gfCNCPoint3[25201] = {X 315.6744, Y 14.7426, Z -4.6667, A 0.000, B 0.000, C 0.000 }
gfCNCPoint3[25202] = {X 315.1915, Y 15.5144, Z -4.6667, A 0.000, B 0.000, C 0.000 }
gfCNCPoint3[25203] = {X 314.5495, Y 16.1599, Z -4.6667, A 0.000, B 0.000, C 0.000 }
gfCNCPoint3[25204] = {X 314.5481, Y 41.0279, Z -4.6667, A 0.000, B 0.000, C 0.000 }
gfCNCPoint3[25205] = {X 314.6336, Y 41.0962, Z -4.6667, A 0.000, B 0.000, C 0.000 }
gfCNCPoint3[25206] = {X 315.2363, Y 41.7299, Z -4.6667, A 0.000, B 0.000, C 0.000 }
gfCNCPoint3[25207] = {X 315.6902, Y 42.4775, Z -4.6667, A 0.000, B 0.000, C 0.000 }
gfCNCPoint3[25208] = {X 315.9743, Y 43.3047, Z -4.6667, A 0.000, B 0.000, C 0.000 }
gfCNCPoint3[25209] = {X 316.0756, Y 44.1734, Z -4.6667, A 0.000, B 0.000, C 0.000 }
gfCNCPoint3[25210] = {X 316.0757, Y 45.0000, Z -4.6667, A 0.000, B 0.000, C 0.000 }
gfCNCPoint3[25211] = {X 315.9734, Y 45.9079, Z -4.6667, A 0.000, B 0.000, C 0.000 }
gfCNCPoint3[25212] = {X 315.6717, Y 46.7702, Z -4.6667, A 0.000, B 0.000, C 0.000 }
gfCNCPoint3[25213] = {X 315.1856, Y 47.5438, Z -4.6667, A 0.000, B 0.000, C 0.000 }
gfCNCPoint3[25214] = {X 314.5396, Y 48.1899, Z -4.6667, A 0.000, B 0.000, C 0.000 }
gfCNCPoint3[25215] = {X 313.7660, Y 48.6760, Z -4.6667, A 0.000, B 0.000, C 0.000 }
gfCNCPoint3[25216] = {X 312.9036, Y 48.9777, Z -4.6667, A 0.000, B 0.000, C 0.000 }
gfCNCPoint3[25217] = {X 311.9957, Y 49.0800, Z -4.6667, A 0.000, B 0.000, C 0.000 }
gfCNCPoint3[25218] = {X 305.5523, Y 49.0800, Z -4.6667, A 0.000, B 0.000, C 0.000 }
gfCNCPoint3[25219] = {X 304.6489, Y 48.9787, Z -4.6667, A 0.000, B 0.000, C 0.000 }
gfCNCPoint3[25220] = {X 303.7905, Y 48.6800, Z -4.6667, A 0.000, B 0.000, C 0.000 }
gfCNCPoint3[25221] = {X 303.0194, Y 48.1986, Z -4.6667, A 0.000, B 0.000, C 0.000 }
gfCNCPoint3[25222] = {X 302.3741, Y 47.5585, Z -4.6667, A 0.000, B 0.000, C 0.000 }
gfCNCPoint3[25223] = {X 301.8865, Y 46.7914, Z -4.6667, A 0.000, B 0.000, C 0.000 }
gfCNCPoint3[25224] = {X 301.5809, Y 45.9353, Z -4.6667, A 0.000, B 0.000, C 0.000 }
gfCNCPoint3[25225] = {X 301.4724, Y 45.0328, Z -4.6667, A 0.000, B 0.000, C 0.000 }
gfCNCPoint3[25226] = {X 301.4723, Y 44.2070, Z -4.6667, A 0.000, B 0.000, C 0.000 }
gfCNCPoint3[25227] = {X 301.5898, Y 43.2934, Z -4.6667, A 0.000, B 0.000, C 0.000 }
gfCNCPoint3[25228] = {X 301.8935, Y 42.4238, Z -4.6667, A 0.000, B 0.000, C 0.000 }
gfCNCPoint3[25229] = {X 302.3704, Y 41.6357, Z -4.6667, A 0.000, B 0.000, C 0.000 }
gfCNCPoint3[25230] = {X 302.9997, Y 40.9632, Z -4.6667, A 0.000, B 0.000, C 0.000 }
gfCNCPoint3[25231] = {X 302.9997, Y 33.7943, Z -4.6667, A 0.000, B 0.000, C 0.000 }
gfCNCPoint3[25232] = {X 293.6145, Y 33.7943, Z -4.6667, A 0.000, B 0.000, C 0.000 }
gfCNCPoint3[25233] = {X 293.6137, Y 41.0139, Z -4.6667, A 0.000, B 0.000, C 0.000 }
gfCNCPoint3[25234] = {X 294.2515, Y 41.6661, Z -4.6667, A 0.000, B 0.000, C 0.000 }
gfCNCPoint3[25235] = {X 294.7325, Y 42.4413, Z -4.6667, A 0.000, B 0.000, C 0.000 }
gfCNCPoint3[25236] = {X 295.0338, Y 43.3023, Z -4.6667, A 0.000, B 0.000, C 0.000 }
gfCNCPoint3[25237] = {X 295.1411, Y 44.2082, Z -4.6667, A 0.000, B 0.000, C 0.000 }
gfCNCPoint3[25238] = {X 295.1411, Y 45.0000, Z -4.6667, A 0.000, B 0.000, C 0.000 }
gfCNCPoint3[25239] = {X 295.0388, Y 45.9079, Z -4.6667, A 0.000, B 0.000, C 0.000 }
gfCNCPoint3[25240] = {X 294.7371, Y 46.7702, Z -4.6667, A 0.000, B 0.000, C 0.000 }
gfCNCPoint3[25241] = {X 294.2510, Y 47.5438, Z -4.6667, A 0.000, B 0.000, C 0.000 }
gfCNCPoint3[25242] = {X 293.6050, Y 48.1899, Z -4.6667, A 0.000, B 0.000, C 0.000 }
gfCNCPoint3[25243] = {X 292.8314, Y 48.6760, Z -4.6667, A 0.000, B 0.000, C 0.000 }
gfCNCPoint3[25244] = {X 291.9690, Y 48.9777, Z -4.6667, A 0.000, B 0.000, C 0.000 }
gfCNCPoint3[25245] = {X 291.0611, Y 49.0800, Z -4.6667, A 0.000, B 0.000, C 0.000 }
gfCNCPoint3[25246] = {X 284.6177, Y 49.0800, Z -4.6667, A 0.000, B 0.000, C 0.000 }
gfCNCPoint3[25247] = {X 283.7144, Y 48.9788, Z -4.6667, A 0.000, B 0.000, C 0.000 }
gfCNCPoint3[25248] = {X 282.8560, Y 48.6801, Z -4.6667, A 0.000, B 0.000, C 0.000 }
gfCNCPoint3[25249] = {X 282.0850, Y 48.1987, Z -4.6667, A 0.000, B 0.000, C 0.000 }
gfCNCPoint3[25250] = {X 281.4397, Y 47.5587, Z -4.6667, A 0.000, B 0.000, C 0.000 }
gfCNCPoint3[25251] = {X 280.9521, Y 46.7916, Z -4.6667, A 0.000, B 0.000, C 0.000 }
gfCNCPoint3[25252] = {X 280.6464, Y 45.9356, Z -4.6667, A 0.000, B 0.000, C 0.000 }
gfCNCPoint3[25253] = {X 280.5378, Y 45.0332, Z -4.6667, A 0.000, B 0.000, C 0.000 }
gfCNCPoint3[25254] = {X 280.5377, Y 44.2085, Z -4.6667, A 0.000, B 0.000, C 0.000 }
gfCNCPoint3[25255] = {X 280.6428, Y 43.3038, Z -4.6667, A 0.000, B 0.000, C 0.000 }
gfCNCPoint3[25256] = {X 280.9436, Y 42.4442, Z -4.6667, A 0.000, B 0.000, C 0.000 }
gfCNCPoint3[25257] = {X 281.4256, Y 41.6715, Z -4.6667, A 0.000, B 0.000, C 0.000 }
gfCNCPoint3[25258] = {X 282.0653, Y 41.0233, Z -4.6667, A 0.000, B 0.000, C 0.000 }
gfCNCPoint3[25259] = {X 282.0651, Y 28.5924, Z -4.6667, A 0.000, B 0.000, C 0.000 }
gfCNCPoint3[25260] = {X 278.0651, Y 28.5925, Z -4.6667, A 0.000, B 0.000, C 0.000 }
gfCNCPoint3[25261] = {X 282.1451, Y 28.5924, Z -4.6667, A 0.000, B 0.000, C 0.000 }
gfCNCPoint3[25262] = {X 282.1449, Y 16.1221, Z -4.6667, A 0.000, B 0.000, C 0.000 }
gfCNCPoint3[25263] = {X 281.5030, Y 15.4878, Z -4.6667, A 0.000, B 0.000, C 0.000 }
gfCNCPoint3[25264] = {X 281.0197, Y 14.7257, Z -4.6667, A 0.000, B 0.000, C 0.000 }
gfCNCPoint3[25265] = {X 280.7195, Y 13.8746, Z -4.6667, A 0.000, B 0.000, C 0.000 }
gfCNCPoint3[25266] = {X 280.6177, Y 12.9779, Z -4.6667, A 0.000, B 0.000, C 0.000 }
gfCNCPoint3[25267] = {X 280.6177, Y 12.1868, Z -4.6667, A 0.000, B 0.000, C 0.000 }
gfCNCPoint3[25268] = {X 280.7180, Y 11.2967, Z -4.6667, A 0.000, B 0.000, C 0.000 }
gfCNCPoint3[25269] = {X 281.0138, Y 10.4513, Z -4.6667, A 0.000, B 0.000, C 0.000 }
gfCNCPoint3[25270] = {X 281.4903, Y 9.6929, Z -4.6667, A 0.000, B 0.000, C 0.000 }
gfCNCPoint3[25271] = {X 282.1237, Y 9.0595, Z -4.6667, A 0.000, B 0.000, C 0.000 }
gfCNCPoint3[25272] = {X 282.8821, Y 8.5829, Z -4.6667, A 0.000, B 0.000, C 0.000 }
gfCNCPoint3[25273] = {X 283.7276, Y 8.2871, Z -4.6667, A 0.000, B 0.000, C 0.000 }
gfCNCPoint3[25274] = {X 284.6177, Y 8.1868, Z -4.6667, A 0.000, B 0.000, C 0.000 }
gfCNCPoint3[25275] = {X 291.0611, Y 8.1868, Z -4.6667, A 0.000, B 0.000, C 0.000 }
gfCNCPoint3[25276] = {X 291.9512, Y 8.2871, Z -4.6667, A 0.000, B 0.000, C 0.000 }
gfCNCPoint3[25277] = {X 292.7967, Y 8.5829, Z -4.6667, A 0.000, B 0.000, C 0.000 }
gfCNCPoint3[25278] = {X 293.5551, Y 9.0595, Z -4.6667, A 0.000, B 0.000, C 0.000 }
gfCNCPoint3[25279] = {X 294.1885, Y 9.6929, Z -4.6667, A 0.000, B 0.000, C 0.000 }
gfCNCPoint3[25280] = {X 294.6650, Y 10.4513, Z -4.6667, A 0.000, B 0.000, C 0.000 }
gfCNCPoint3[25281] = {X 294.9608, Y 11.2967, Z -4.6667, A 0.000, B 0.000, C 0.000 }
gfCNCPoint3[25282] = {X 295.0611, Y 12.1868, Z -4.6667, A 0.000, B 0.000, C 0.000 }
gfCNCPoint3[25283] = {X 295.0609, Y 13.0192, Z -4.6667, A 0.000, B 0.000, C 0.000 }
gfCNCPoint3[25284] = {X 294.9625, Y 13.8611, Z -4.6667, A 0.000, B 0.000, C 0.000 }
gfCNCPoint3[25285] = {X 294.6888, Y 14.6633, Z -4.6667, A 0.000, B 0.000, C 0.000 }
gfCNCPoint3[25286] = {X 294.2523, Y 15.3898, Z -4.6667, A 0.000, B 0.000, C 0.000 }
gfCNCPoint3[25287] = {X 293.6725, Y 16.0080, Z -4.6667, A 0.000, B 0.000, C 0.000 }
gfCNCPoint3[25288] = {X 293.5959, Y 16.0724, Z -4.6667, A 0.000, B 0.000, C 0.000 }
gfCNCPoint3[25289] = {X 293.5177, Y 16.1348, Z -4.6667, A 0.000, B 0.000, C 0.000 }
gfCNCPoint3[25290] = {X 293.5336, Y 16.1923, Z -4.6667, A 0.000, B 0.000, C 0.000 }
gfCNCPoint3[25291] = {X 293.5348, Y 22.5166, Z -4.6667, A 0.000, B 0.000, C 0.000 }
gfCNCPoint3[25292] = {X 293.7676, Y 22.5165, Z -4.6667, A 0.000, B 0.000, C 0.000 }
gfCNCPoint3[25293] = {X 303.0789, Y 22.5170, Z -4.6667, A 0.000, B 0.000, C 0.000 }
gfCNCPoint3[25294] = {X 303.0794, Y 16.1925, Z -4.6667, A 0.000, B 0.000, C 0.000 }
gfCNCPoint3[25295] = {X 303.0955, Y 16.1346, Z -4.6667, A 0.000, B 0.000, C 0.000 }
gfCNCPoint3[25296] = {X 303.0172, Y 16.0722, Z -4.6667, A 0.000, B 0.000, C 0.000 }
gfCNCPoint3[25297] = {X 302.9406, Y 16.0077, Z -4.6667, A 0.000, B 0.000, C 0.000 }
gfCNCPoint3[25298] = {X 302.3547, Y 15.3813, Z -4.6667, A 0.000, B 0.000, C 0.000 }
gfCNCPoint3[25299] = {X 301.9158, Y 14.6443, Z -4.6667, A 0.000, B 0.000, C 0.000 }
gfCNCPoint3[25300] = {X 301.6442, Y 13.8307, Z -4.6667, A 0.000, B 0.000, C 0.000 }
gfCNCPoint3[25301] = {X 301.5523, Y 12.9779, Z -4.6667, A 0.000, B 0.000, C 0.000 }
gfCNCPoint3[25302] = {X 301.5523, Y 12.1868, Z -4.6667, A 0.000, B 0.000, C 0.000 }
gfCNCPoint3[25303] = {X 301.6525, Y 11.2967, Z -4.6667, A 0.000, B 0.000, C 0.000 }
gfCNCPoint3[25304] = {X 301.9484, Y 10.4513, Z -4.6667, A 0.000, B 0.000, C 0.000 }
gfCNCPoint3[25305] = {X 302.4249, Y 9.6929, Z -4.6667, A 0.000, B 0.000, C 0.000 }
gfCNCPoint3[25306] = {X 303.0583, Y 9.0595, Z -4.6667, A 0.000, B 0.000, C 0.000 }
gfCNCPoint3[25307] = {X 303.8167, Y 8.5829, Z -4.6667, A 0.000, B 0.000, C 0.000 }
gfCNCPoint3[25308] = {X 304.6622, Y 8.2871, Z -4.6667, A 0.000, B 0.000, C 0.000 }
gfCNCPoint3[25309] = {X 305.5523, Y 8.1868, Z -4.6667, A 0.000, B 0.000, C 0.000 }
gfCNCPoint3[25310] = {X 311.9957, Y 8.1868, Z -4.6667, A 0.000, B 0.000, C 0.000 }
gfCNCPoint3[25311] = {X 312.8858, Y 8.2871, Z -4.6667, A 0.000, B 0.000, C 0.000 }
gfCNCPoint3[25312] = {X 313.7313, Y 8.5829, Z -4.6667, A 0.000, B 0.000, C 0.000 }
gfCNCPoint3[25313] = {X 314.4897, Y 9.0595, Z -4.6667, A 0.000, B 0.000, C 0.000 }
gfCNCPoint3[25314] = {X 315.1230, Y 9.6929, Z -4.6667, A 0.000, B 0.000, C 0.000 }
gfCNCPoint3[25315] = {X 315.5996, Y 10.4513, Z -4.6667, A 0.000, B 0.000, C 0.000 }
gfCNCPoint3[25316] = {X 315.8954, Y 11.2967, Z -4.6667, A 0.000, B 0.000, C 0.000 }
gfCNCPoint3[25317] = {X 315.9957, Y 12.1868, Z -4.6667, A 0.000, B 0.000, C 0.000 }
gfCNCPoint3[25318] = {X 315.9955, Y 13.0192, Z -4.6667, A 0.000, B 0.000, C 0.000 }
gfCNCPoint3[25319] = {X 315.8870, Y 13.9044, Z -4.6667, A 0.000, B 0.000, C 0.000 }
gfCNCPoint3[25320] = {X 315.5850, Y 14.7436, Z -4.6667, A 0.000, B 0.000, C 0.000 }
gfCNCPoint3[25321] = {X 315.1045, Y 15.4950, Z -4.6667, A 0.000, B 0.000, C 0.000 }
gfCNCPoint3[25322] = {X 314.4695, Y 16.1213, Z -4.6667, A 0.000, B 0.000, C 0.000 }
gfCNCPoint3[25323] = {X 314.4681, Y 41.0664, Z -4.6667, A 0.000, B 0.000, C 0.000 }
gfCNCPoint3[25324] = {X 314.6070, Y 41.1787, Z -4.6667, A 0.000, B 0.000, C 0.000 }
gfCNCPoint3[25325] = {X 315.1930, Y 41.8052, Z -4.6667, A 0.000, B 0.000, C 0.000 }
gfCNCPoint3[25326] = {X 315.6320, Y 42.5423, Z -4.6667, A 0.000, B 0.000, C 0.000 }
gfCNCPoint3[25327] = {X 315.9038, Y 43.3560, Z -4.6667, A 0.000, B 0.000, C 0.000 }
gfCNCPoint3[25328] = {X 315.9957, Y 44.2089, Z -4.6667, A 0.000, B 0.000, C 0.000 }
gfCNCPoint3[25329] = {X 315.9957, Y 45.0000, Z -4.6667, A 0.000, B 0.000, C 0.000 }
gfCNCPoint3[25330] = {X 315.8954, Y 45.8901, Z -4.6667, A 0.000, B 0.000, C 0.000 }
gfCNCPoint3[25331] = {X 315.5996, Y 46.7355, Z -4.6667, A 0.000, B 0.000, C 0.000 }
gfCNCPoint3[25332] = {X 315.1230, Y 47.4940, Z -4.6667, A 0.000, B 0.000, C 0.000 }
gfCNCPoint3[25333] = {X 314.4897, Y 48.1273, Z -4.6667, A 0.000, B 0.000, C 0.000 }
gfCNCPoint3[25334] = {X 313.7313, Y 48.6039, Z -4.6667, A 0.000, B 0.000, C 0.000 }
gfCNCPoint3[25335] = {X 312.8858, Y 48.8997, Z -4.6667, A 0.000, B 0.000, C 0.000 }
gfCNCPoint3[25336] = {X 311.9957, Y 49.0000, Z -4.6667, A 0.000, B 0.000, C 0.000 }
gfCNCPoint3[25337] = {X 305.5523, Y 49.0000, Z -4.6667, A 0.000, B 0.000, C 0.000 }
gfCNCPoint3[25338] = {X 304.6622, Y 48.8997, Z -4.6667, A 0.000, B 0.000, C 0.000 }
gfCNCPoint3[25339] = {X 303.8167, Y 48.6039, Z -4.6667, A 0.000, B 0.000, C 0.000 }
gfCNCPoint3[25340] = {X 303.0583, Y 48.1273, Z -4.6667, A 0.000, B 0.000, C 0.000 }
gfCNCPoint3[25341] = {X 302.4249, Y 47.4939, Z -4.6667, A 0.000, B 0.000, C 0.000 }
gfCNCPoint3[25342] = {X 301.9484, Y 46.7355, Z -4.6667, A 0.000, B 0.000, C 0.000 }
gfCNCPoint3[25343] = {X 301.6525, Y 45.8901, Z -4.6667, A 0.000, B 0.000, C 0.000 }
gfCNCPoint3[25344] = {X 301.5523, Y 45.0000, Z -4.6667, A 0.000, B 0.000, C 0.000 }
gfCNCPoint3[25345] = {X 301.5523, Y 44.2089, Z -4.6667, A 0.000, B 0.000, C 0.000 }
gfCNCPoint3[25346] = {X 301.6698, Y 43.3029, Z -4.6667, A 0.000, B 0.000, C 0.000 }
gfCNCPoint3[25347] = {X 301.9737, Y 42.4414, Z -4.6667, A 0.000, B 0.000, C 0.000 }
gfCNCPoint3[25348] = {X 302.4507, Y 41.6623, Z -4.6667, A 0.000, B 0.000, C 0.000 }
gfCNCPoint3[25349] = {X 303.0797, Y 40.9999, Z -4.6667, A 0.000, B 0.000, C 0.000 }
gfCNCPoint3[25350] = {X 303.0797, Y 33.7143, Z -4.6667, A 0.000, B 0.000, C 0.000 }
gfCNCPoint3[25351] = {X 293.9345, Y 33.7143, Z -4.6667, A 0.000, B 0.000, C 0.000 }
gfCNCPoint3[25352] = {X 293.5345, Y 33.7139, Z -4.6667, A 0.000, B 0.000, C 0.000 }
gfCNCPoint3[25353] = {X 293.5337, Y 41.0520, Z -4.6667, A 0.000, B 0.000, C 0.000 }
gfCNCPoint3[25354] = {X 294.1710, Y 41.6933, Z -4.6667, A 0.000, B 0.000, C 0.000 }
gfCNCPoint3[25355] = {X 294.6521, Y 42.4588, Z -4.6667, A 0.000, B 0.000, C 0.000 }
gfCNCPoint3[25356] = {X 294.9538, Y 43.3111, Z -4.6667, A 0.000, B 0.000, C 0.000 }
gfCNCPoint3[25357] = {X 295.0611, Y 44.2089, Z -4.6667, A 0.000, B 0.000, C 0.000 }
gfCNCPoint3[25358] = {X 295.0611, Y 45.0000, Z -4.6667, A 0.000, B 0.000, C 0.000 }
gfCNCPoint3[25359] = {X 294.9608, Y 45.8901, Z -4.6667, A 0.000, B 0.000, C 0.000 }
gfCNCPoint3[25360] = {X 294.6650, Y 46.7355, Z -4.6667, A 0.000, B 0.000, C 0.000 }
gfCNCPoint3[25361] = {X 294.1885, Y 47.4940, Z -4.6667, A 0.000, B 0.000, C 0.000 }
gfCNCPoint3[25362] = {X 293.5551, Y 48.1273, Z -4.6667, A 0.000, B 0.000, C 0.000 }
gfCNCPoint3[25363] = {X 292.7967, Y 48.6039, Z -4.6667, A 0.000, B 0.000, C 0.000 }
gfCNCPoint3[25364] = {X 291.9512, Y 48.8997, Z -4.6667, A 0.000, B 0.000, C 0.000 }
gfCNCPoint3[25365] = {X 291.0611, Y 49.0000, Z -4.6667, A 0.000, B 0.000, C 0.000 }
gfCNCPoint3[25366] = {X 284.6177, Y 49.0000, Z -4.6667, A 0.000, B 0.000, C 0.000 }
gfCNCPoint3[25367] = {X 283.7276, Y 48.8997, Z -4.6667, A 0.000, B 0.000, C 0.000 }
gfCNCPoint3[25368] = {X 282.8821, Y 48.6039, Z -4.6667, A 0.000, B 0.000, C 0.000 }
gfCNCPoint3[25369] = {X 282.1237, Y 48.1273, Z -4.6667, A 0.000, B 0.000, C 0.000 }
gfCNCPoint3[25370] = {X 281.4903, Y 47.4939, Z -4.6667, A 0.000, B 0.000, C 0.000 }
gfCNCPoint3[25371] = {X 281.0138, Y 46.7355, Z -4.6667, A 0.000, B 0.000, C 0.000 }
gfCNCPoint3[25372] = {X 280.7180, Y 45.8901, Z -4.6667, A 0.000, B 0.000, C 0.000 }
gfCNCPoint3[25373] = {X 280.6177, Y 45.0000, Z -4.6667, A 0.000, B 0.000, C 0.000 }
gfCNCPoint3[25374] = {X 280.6177, Y 44.2089, Z -4.6667, A 0.000, B 0.000, C 0.000 }
gfCNCPoint3[25375] = {X 280.7229, Y 43.3125, Z -4.6667, A 0.000, B 0.000, C 0.000 }
gfCNCPoint3[25376] = {X 281.0240, Y 42.4617, Z -4.6667, A 0.000, B 0.000, C 0.000 }
gfCNCPoint3[25377] = {X 281.5062, Y 41.6988, Z -4.6667, A 0.000, B 0.000, C 0.000 }
gfCNCPoint3[25378] = {X 282.1453, Y 41.0616, Z -4.6667, A 0.000, B 0.000, C 0.000 }
gfCNCPoint3[25379] = {X 282.1451, Y 28.5924, Z -4.6667, A 0.000, B 0.000, C 0.000 }
gfCNCPoint3[25380] = {X 278.0651, Y 28.5925, Z -4.6667, A 0.000, B 0.000, C 0.000 }
gfCNCPoint3[25381] = {X 278.0651, Y 28.5925, Z -1.6667, A 0.000, B 0.000, C 0.000 }
gfCNCPoint3[25382] = {X 278.0651, Y 28.5925, Z 11.0000, A 0.000, B 0.000, C 0.000 }
gfCNCPoint3[25383] = {X 353.3541, Y 107.0405, Z 11.0000, A 0.000, B 0.000, C 0.000 }
gfCNCPoint3[25384] = {X 353.3541, Y 107.0405, Z -1.6667, A 0.000, B 0.000, C 0.000 }
gfCNCPoint3[25385] = {X 353.3541, Y 107.0405, Z -4.6667, A 0.000, B 0.000, C 0.000 }
gfCNCPoint3[25386] = {X 353.2427, Y 102.9621, Z -4.6667, A 0.000, B 0.000, C 0.000 }
gfCNCPoint3[25387] = {X 348.1840, Y 103.0319, Z -4.6667, A 0.000, B 0.000, C 0.000 }
gfCNCPoint3[25388] = {X 343.1252, Y 102.9652, Z -4.6667, A 0.000, B 0.000, C 0.000 }
gfCNCPoint3[25389] = {X 338.0701, Y 102.7618, Z -4.6667, A 0.000, B 0.000, C 0.000 }
gfCNCPoint3[25390] = {X 334.1158, Y 102.4849, Z -4.6667, A 0.000, B 0.000, C 0.000 }
gfCNCPoint3[25391] = {X 330.1765, Y 102.0430, Z -4.6667, A 0.000, B 0.000, C 0.000 }
gfCNCPoint3[25392] = {X 326.2591, Y 101.4370, Z -4.6667, A 0.000, B 0.000, C 0.000 }
gfCNCPoint3[25393] = {X 323.4092, Y 100.8331, Z -4.6667, A 0.000, B 0.000, C 0.000 }
gfCNCPoint3[25394] = {X 320.6117, Y 100.0201, Z -4.6667, A 0.000, B 0.000, C 0.000 }
gfCNCPoint3[25395] = {X 317.8820, Y 99.0025, Z -4.6667, A 0.000, B 0.000, C 0.000 }
gfCNCPoint3[25396] = {X 316.3696, Y 98.3039, Z -4.6667, A 0.000, B 0.000, C 0.000 }
gfCNCPoint3[25397] = {X 314.9207, Y 97.4819, Z -4.6667, A 0.000, B 0.000, C 0.000 }
gfCNCPoint3[25398] = {X 313.5452, Y 96.5421, Z -4.6667, A 0.000, B 0.000, C 0.000 }
gfCNCPoint3[25399] = {X 312.2527, Y 95.4911, Z -4.6667, A 0.000, B 0.000, C 0.000 }
gfCNCPoint3[25400] = {X 311.2489, Y 94.4926, Z -4.6667, A 0.000, B 0.000, C 0.000 }
gfCNCPoint3[25401] = {X 310.3706, Y 93.3822, Z -4.6667, A 0.000, B 0.000, C 0.000 }
gfCNCPoint3[25402] = {X 309.6302, Y 92.1754, Z -4.6667, A 0.000, B 0.000, C 0.000 }
gfCNCPoint3[25403] = {X 309.0381, Y 90.8894, Z -4.6667, A 0.000, B 0.000, C 0.000 }
gfCNCPoint3[25404] = {X 308.6026, Y 89.5423, Z -4.6667, A 0.000, B 0.000, C 0.000 }
gfCNCPoint3[25405] = {X 308.2592, Y 87.9192, Z -4.6667, A 0.000, B 0.000, C 0.000 }
gfCNCPoint3[25406] = {X 308.0563, Y 86.2726, Z -4.6667, A 0.000, B 0.000, C 0.000 }
gfCNCPoint3[25407] = {X 307.9954, Y 84.6147, Z -4.6667, A 0.000, B 0.000, C 0.000 }
gfCNCPoint3[25408] = {X 307.9966, Y 63.2123, Z -4.6667, A 0.000, B 0.000, C 0.000 }
gfCNCPoint3[25409] = {X 307.1451, Y 63.0030, Z -4.6667, A 0.000, B 0.000, C 0.000 }
gfCNCPoint3[25410] = {X 306.3533, Y 62.6262, Z -4.6667, A 0.000, B 0.000, C 0.000 }
gfCNCPoint3[25411] = {X 305.6540, Y 62.0972, Z -4.6667, A 0.000, B 0.000, C 0.000 }
gfCNCPoint3[25412] = {X 305.0759, Y 61.4379, Z -4.6667, A 0.000, B 0.000, C 0.000 }
gfCNCPoint3[25413] = {X 304.6428, Y 60.6755, Z -4.6667, A 0.000, B 0.000, C 0.000 }
gfCNCPoint3[25414] = {X 304.3726, Y 59.8413, Z -4.6667, A 0.000, B 0.000, C 0.000 }
gfCNCPoint3[25415] = {X 304.2764, Y 58.9697, Z -4.6667, A 0.000, B 0.000, C 0.000 }
gfCNCPoint3[25416] = {X 304.2762, Y 58.0000, Z -4.6667, A 0.000, B 0.000, C 0.000 }
gfCNCPoint3[25417] = {X 304.3845, Y 57.0387, Z -4.6667, A 0.000, B 0.000, C 0.000 }
gfCNCPoint3[25418] = {X 304.7040, Y 56.1256, Z -4.6667, A 0.000, B 0.000, C 0.000 }
gfCNCPoint3[25419] = {X 305.2187, Y 55.3065, Z -4.6667, A 0.000, B 0.000, C 0.000 }
gfCNCPoint3[25420] = {X 305.9027, Y 54.6225, Z -4.6667, A 0.000, B 0.000, C 0.000 }
gfCNCPoint3[25421] = {X 306.7218, Y 54.1078, Z -4.6667, A 0.000, B 0.000, C 0.000 }
gfCNCPoint3[25422] = {X 307.6349, Y 53.7883, Z -4.6667, A 0.000, B 0.000, C 0.000 }
gfCNCPoint3[25423] = {X 308.5962, Y 53.6800, Z -4.6667, A 0.000, B 0.000, C 0.000 }
gfCNCPoint3[25424] = {X 324.3107, Y 53.6800, Z -4.6667, A 0.000, B 0.000, C 0.000 }
gfCNCPoint3[25425] = {X 325.2720, Y 53.7883, Z -4.6667, A 0.000, B 0.000, C 0.000 }
gfCNCPoint3[25426] = {X 326.1851, Y 54.1078, Z -4.6667, A 0.000, B 0.000, C 0.000 }
gfCNCPoint3[25427] = {X 327.0042, Y 54.6225, Z -4.6667, A 0.000, B 0.000, C 0.000 }
gfCNCPoint3[25428] = {X 327.6882, Y 55.3065, Z -4.6667, A 0.000, B 0.000, C 0.000 }
gfCNCPoint3[25429] = {X 328.2029, Y 56.1256, Z -4.6667, A 0.000, B 0.000, C 0.000 }
gfCNCPoint3[25430] = {X 328.5224, Y 57.0387, Z -4.6667, A 0.000, B 0.000, C 0.000 }
gfCNCPoint3[25431] = {X 328.6307, Y 58.0000, Z -4.6667, A 0.000, B 0.000, C 0.000 }
gfCNCPoint3[25432] = {X 328.6307, Y 58.9359, Z -4.6667, A 0.000, B 0.000, C 0.000 }
gfCNCPoint3[25433] = {X 328.5366, Y 59.8122, Z -4.6667, A 0.000, B 0.000, C 0.000 }
gfCNCPoint3[25434] = {X 328.2681, Y 60.6516, Z -4.6667, A 0.000, B 0.000, C 0.000 }
gfCNCPoint3[25435] = {X 327.8362, Y 61.4199, Z -4.6667, A 0.000, B 0.000, C 0.000 }
gfCNCPoint3[25436] = {X 327.2587, Y 62.0856, Z -4.6667, A 0.000, B 0.000, C 0.000 }
gfCNCPoint3[25437] = {X 326.5590, Y 62.6214, Z -4.6667, A 0.000, B 0.000, C 0.000 }
gfCNCPoint3[25438] = {X 325.7658, Y 63.0056, Z -4.6667, A 0.000, B 0.000, C 0.000 }
gfCNCPoint3[25439] = {X 324.9116, Y 63.2223, Z -4.6667, A 0.000, B 0.000, C 0.000 }
gfCNCPoint3[25440] = {X 324.9132, Y 83.2295, Z -4.6667, A 0.000, B 0.000, C 0.000 }
gfCNCPoint3[25441] = {X 324.9268, Y 84.6147, Z -4.6667, A 0.000, B 0.000, C 0.000 }
gfCNCPoint3[25442] = {X 325.0042, Y 85.8499, Z -4.6667, A 0.000, B 0.000, C 0.000 }
gfCNCPoint3[25443] = {X 325.2261, Y 87.0674, Z -4.6667, A 0.000, B 0.000, C 0.000 }
gfCNCPoint3[25444] = {X 325.4715, Y 87.3361, Z -4.6667, A 0.000, B 0.000, C 0.000 }
gfCNCPoint3[25445] = {X 325.7737, Y 87.5389, Z -4.6667, A 0.000, B 0.000, C 0.000 }
gfCNCPoint3[25446] = {X 326.2246, Y 87.7937, Z -4.6667, A 0.000, B 0.000, C 0.000 }
gfCNCPoint3[25447] = {X 327.6624, Y 88.3904, Z -4.6667, A 0.000, B 0.000, C 0.000 }
gfCNCPoint3[25448] = {X 329.1569, Y 88.8260, Z -4.6667, A 0.000, B 0.000, C 0.000 }
gfCNCPoint3[25449] = {X 332.2329, Y 89.4419, Z -4.6667, A 0.000, B 0.000, C 0.000 }
gfCNCPoint3[25450] = {X 335.3453, Y 89.8349, Z -4.6667, A 0.000, B 0.000, C 0.000 }
gfCNCPoint3[25451] = {X 339.4834, Y 90.1549, Z -4.6667, A 0.000, B 0.000, C 0.000 }
gfCNCPoint3[25452] = {X 343.6300, Y 90.3344, Z -4.6667, A 0.000, B 0.000, C 0.000 }
gfCNCPoint3[25453] = {X 347.7803, Y 90.3734, Z -4.6667, A 0.000, B 0.000, C 0.000 }
gfCNCPoint3[25454] = {X 352.1620, Y 90.3350, Z -4.6667, A 0.000, B 0.000, C 0.000 }
gfCNCPoint3[25455] = {X 356.5395, Y 90.1391, Z -4.6667, A 0.000, B 0.000, C 0.000 }
gfCNCPoint3[25456] = {X 360.9071, Y 89.7860, Z -4.6667, A 0.000, B 0.000, C 0.000 }
gfCNCPoint3[25457] = {X 363.2212, Y 89.4982, Z -4.6667, A 0.000, B 0.000, C 0.000 }
gfCNCPoint3[25458] = {X 365.5139, Y 89.0719, Z -4.6667, A 0.000, B 0.000, C 0.000 }
gfCNCPoint3[25459] = {X 367.7768, Y 88.5085, Z -4.6667, A 0.000, B 0.000, C 0.000 }
gfCNCPoint3[25460] = {X 368.7087, Y 88.1952, Z -4.6667, A 0.000, B 0.000, C 0.000 }
gfCNCPoint3[25461] = {X 369.5996, Y 87.7794, Z -4.6667, A 0.000, B 0.000, C 0.000 }
gfCNCPoint3[25462] = {X 370.4383, Y 87.2663, Z -4.6667, A 0.000, B 0.000, C 0.000 }
gfCNCPoint3[25463] = {X 370.5880, Y 87.1105, Z -4.6667, A 0.000, B 0.000, C 0.000 }
gfCNCPoint3[25464] = {X 370.6652, Y 86.9086, Z -4.6667, A 0.000, B 0.000, C 0.000 }
gfCNCPoint3[25465] = {X 370.8563, Y 85.3737, Z -4.6667, A 0.000, B 0.000, C 0.000 }
gfCNCPoint3[25466] = {X 370.9201, Y 83.8283, Z -4.6667, A 0.000, B 0.000, C 0.000 }
gfCNCPoint3[25467] = {X 370.9205, Y 63.2124, Z -4.6667, A 0.000, B 0.000, C 0.000 }
gfCNCPoint3[25468] = {X 370.0688, Y 63.0033, Z -4.6667, A 0.000, B 0.000, C 0.000 }
gfCNCPoint3[25469] = {X 369.2769, Y 62.6265, Z -4.6667, A 0.000, B 0.000, C 0.000 }
gfCNCPoint3[25470] = {X 368.5774, Y 62.0975, Z -4.6667, A 0.000, B 0.000, C 0.000 }
gfCNCPoint3[25471] = {X 367.9991, Y 61.4382, Z -4.6667, A 0.000, B 0.000, C 0.000 }
gfCNCPoint3[25472] = {X 367.5659, Y 60.6757, Z -4.6667, A 0.000, B 0.000, C 0.000 }
gfCNCPoint3[25473] = {X 367.2956, Y 59.8414, Z -4.6667, A 0.000, B 0.000, C 0.000 }
gfCNCPoint3[25474] = {X 367.1994, Y 58.9697, Z -4.6667, A 0.000, B 0.000, C 0.000 }
gfCNCPoint3[25475] = {X 367.1993, Y 58.0000, Z -4.6667, A 0.000, B 0.000, C 0.000 }
gfCNCPoint3[25476] = {X 367.3076, Y 57.0387, Z -4.6667, A 0.000, B 0.000, C 0.000 }
gfCNCPoint3[25477] = {X 367.6271, Y 56.1256, Z -4.6667, A 0.000, B 0.000, C 0.000 }
gfCNCPoint3[25478] = {X 368.1418, Y 55.3065, Z -4.6667, A 0.000, B 0.000, C 0.000 }
gfCNCPoint3[25479] = {X 368.8258, Y 54.6225, Z -4.6667, A 0.000, B 0.000, C 0.000 }
gfCNCPoint3[25480] = {X 369.6449, Y 54.1078, Z -4.6667, A 0.000, B 0.000, C 0.000 }
gfCNCPoint3[25481] = {X 370.5580, Y 53.7883, Z -4.6667, A 0.000, B 0.000, C 0.000 }
gfCNCPoint3[25482] = {X 371.5193, Y 53.6800, Z -4.6667, A 0.000, B 0.000, C 0.000 }
gfCNCPoint3[25483] = {X 388.0597, Y 53.6800, Z -4.6667, A 0.000, B 0.000, C 0.000 }
gfCNCPoint3[25484] = {X 389.0210, Y 53.7883, Z -4.6667, A 0.000, B 0.000, C 0.000 }
gfCNCPoint3[25485] = {X 389.9341, Y 54.1078, Z -4.6667, A 0.000, B 0.000, C 0.000 }
gfCNCPoint3[25486] = {X 390.7532, Y 54.6225, Z -4.6667, A 0.000, B 0.000, C 0.000 }
gfCNCPoint3[25487] = {X 391.4372, Y 55.3065, Z -4.6667, A 0.000, B 0.000, C 0.000 }
gfCNCPoint3[25488] = {X 391.9519, Y 56.1256, Z -4.6667, A 0.000, B 0.000, C 0.000 }
gfCNCPoint3[25489] = {X 392.2714, Y 57.0387, Z -4.6667, A 0.000, B 0.000, C 0.000 }
gfCNCPoint3[25490] = {X 392.3797, Y 58.0000, Z -4.6667, A 0.000, B 0.000, C 0.000 }
gfCNCPoint3[25491] = {X 392.3797, Y 58.9342, Z -4.6667, A 0.000, B 0.000, C 0.000 }
gfCNCPoint3[25492] = {X 392.2660, Y 59.9188, Z -4.6667, A 0.000, B 0.000, C 0.000 }
gfCNCPoint3[25493] = {X 391.9308, Y 60.8515, Z -4.6667, A 0.000, B 0.000, C 0.000 }
gfCNCPoint3[25494] = {X 391.4879, Y 61.5648, Z -4.6667, A 0.000, B 0.000, C 0.000 }
gfCNCPoint3[25495] = {X 390.9159, Y 62.1796, Z -4.6667, A 0.000, B 0.000, C 0.000 }
gfCNCPoint3[25496] = {X 390.2363, Y 62.6728, Z -4.6667, A 0.000, B 0.000, C 0.000 }
gfCNCPoint3[25497] = {X 389.4745, Y 63.0259, Z -4.6667, A 0.000, B 0.000, C 0.000 }
gfCNCPoint3[25498] = {X 388.6590, Y 63.2259, Z -4.6667, A 0.000, B 0.000, C 0.000 }
gfCNCPoint3[25499] = {X 388.6569, Y 84.6147, Z -4.6667, A 0.000, B 0.000, C 0.000 }
gfCNCPoint3[25500] = {X 388.5970, Y 86.2730, Z -4.6667, A 0.000, B 0.000, C 0.000 }
gfCNCPoint3[25501] = {X 388.3927, Y 87.9198, Z -4.6667, A 0.000, B 0.000, C 0.000 }
gfCNCPoint3[25502] = {X 388.0455, Y 89.5426, Z -4.6667, A 0.000, B 0.000, C 0.000 }
gfCNCPoint3[25503] = {X 387.5133, Y 91.1299, Z -4.6667, A 0.000, B 0.000, C 0.000 }
gfCNCPoint3[25504] = {X 386.7638, Y 92.6268, Z -4.6667, A 0.000, B 0.000, C 0.000 }
gfCNCPoint3[25505] = {X 385.8117, Y 94.0039, Z -4.6667, A 0.000, B 0.000, C 0.000 }
gfCNCPoint3[25506] = {X 384.6758, Y 95.2338, Z -4.6667, A 0.000, B 0.000, C 0.000 }
gfCNCPoint3[25507] = {X 383.1614, Y 96.5099, Z -4.6667, A 0.000, B 0.000, C 0.000 }
gfCNCPoint3[25508] = {X 381.5201, Y 97.6180, Z -4.6667, A 0.000, B 0.000, C 0.000 }
gfCNCPoint3[25509] = {X 379.7703, Y 98.5456, Z -4.6667, A 0.000, B 0.000, C 0.000 }
gfCNCPoint3[25510] = {X 377.4991, Y 99.5017, Z -4.6667, A 0.000, B 0.000, C 0.000 }
gfCNCPoint3[25511] = {X 375.1651, Y 100.2920, Z -4.6667, A 0.000, B 0.000, C 0.000 }
gfCNCPoint3[25512] = {X 372.7802, Y 100.9123, Z -4.6667, A 0.000, B 0.000, C 0.000 }
gfCNCPoint3[25513] = {X 368.8695, Y 101.6664, Z -4.6667, A 0.000, B 0.000, C 0.000 }
gfCNCPoint3[25514] = {X 364.9264, Y 102.2267, Z -4.6667, A 0.000, B 0.000, C 0.000 }
gfCNCPoint3[25515] = {X 360.9605, Y 102.5918, Z -4.6667, A 0.000, B 0.000, C 0.000 }
gfCNCPoint3[25516] = {X 357.1035, Y 102.8167, Z -4.6667, A 0.000, B 0.000, C 0.000 }
gfCNCPoint3[25517] = {X 353.2427, Y 102.9621, Z -4.6667, A 0.000, B 0.000, C 0.000 }
gfCNCPoint3[25518] = {X 353.3519, Y 106.9606, Z -4.6667, A 0.000, B 0.000, C 0.000 }
gfCNCPoint3[25519] = {X 353.2405, Y 102.8821, Z -4.6667, A 0.000, B 0.000, C 0.000 }
gfCNCPoint3[25520] = {X 348.1839, Y 102.9519, Z -4.6667, A 0.000, B 0.000, C 0.000 }
gfCNCPoint3[25521] = {X 343.1272, Y 102.8852, Z -4.6667, A 0.000, B 0.000, C 0.000 }
gfCNCPoint3[25522] = {X 338.0742, Y 102.6819, Z -4.6667, A 0.000, B 0.000, C 0.000 }
gfCNCPoint3[25523] = {X 334.1232, Y 102.4052, Z -4.6667, A 0.000, B 0.000, C 0.000 }
gfCNCPoint3[25524] = {X 330.1871, Y 101.9637, Z -4.6667, A 0.000, B 0.000, C 0.000 }
gfCNCPoint3[25525] = {X 326.2729, Y 101.3582, Z -4.6667, A 0.000, B 0.000, C 0.000 }
gfCNCPoint3[25526] = {X 323.4287, Y 100.7555, Z -4.6667, A 0.000, B 0.000, C 0.000 }
gfCNCPoint3[25527] = {X 320.6369, Y 99.9442, Z -4.6667, A 0.000, B 0.000, C 0.000 }
gfCNCPoint3[25528] = {X 317.9126, Y 98.9286, Z -4.6667, A 0.000, B 0.000, C 0.000 }
gfCNCPoint3[25529] = {X 316.4063, Y 98.2328, Z -4.6667, A 0.000, B 0.000, C 0.000 }
gfCNCPoint3[25530] = {X 314.9631, Y 97.4140, Z -4.6667, A 0.000, B 0.000, C 0.000 }
gfCNCPoint3[25531] = {X 313.5931, Y 96.4780, Z -4.6667, A 0.000, B 0.000, C 0.000 }
gfCNCPoint3[25532] = {X 312.3057, Y 95.4312, Z -4.6667, A 0.000, B 0.000, C 0.000 }
gfCNCPoint3[25533] = {X 311.3086, Y 94.4394, Z -4.6667, A 0.000, B 0.000, C 0.000 }
gfCNCPoint3[25534] = {X 310.4362, Y 93.3364, Z -4.6667, A 0.000, B 0.000, C 0.000 }
gfCNCPoint3[25535] = {X 309.7008, Y 92.1378, Z -4.6667, A 0.000, B 0.000, C 0.000 }
gfCNCPoint3[25536] = {X 309.1126, Y 90.8604, Z -4.6667, A 0.000, B 0.000, C 0.000 }
gfCNCPoint3[25537] = {X 308.6801, Y 89.5222, Z -4.6667, A 0.000, B 0.000, C 0.000 }
gfCNCPoint3[25538] = {X 308.3380, Y 87.9058, Z -4.6667, A 0.000, B 0.000, C 0.000 }
gfCNCPoint3[25539] = {X 308.1360, Y 86.2660, Z -4.6667, A 0.000, B 0.000, C 0.000 }
gfCNCPoint3[25540] = {X 308.0754, Y 84.6150, Z -4.6667, A 0.000, B 0.000, C 0.000 }
gfCNCPoint3[25541] = {X 308.0766, Y 63.1421, Z -4.6667, A 0.000, B 0.000, C 0.000 }
gfCNCPoint3[25542] = {X 307.2282, Y 62.9473, Z -4.6667, A 0.000, B 0.000, C 0.000 }
gfCNCPoint3[25543] = {X 306.4374, Y 62.5833, Z -4.6667, A 0.000, B 0.000, C 0.000 }
gfCNCPoint3[25544] = {X 305.7377, Y 62.0656, Z -4.6667, A 0.000, B 0.000, C 0.000 }
gfCNCPoint3[25545] = {X 305.1584, Y 61.4158, Z -4.6667, A 0.000, B 0.000, C 0.000 }
gfCNCPoint3[25546] = {X 304.7240, Y 60.6614, Z -4.6667, A 0.000, B 0.000, C 0.000 }
gfCNCPoint3[25547] = {X 304.4529, Y 59.8342, Z -4.6667, A 0.000, B 0.000, C 0.000 }
gfCNCPoint3[25548] = {X 304.3564, Y 58.9691, Z -4.6667, A 0.000, B 0.000, C 0.000 }
gfCNCPoint3[25549] = {X 304.3562, Y 58.0000, Z -4.6667, A 0.000, B 0.000, C 0.000 }
gfCNCPoint3[25550] = {X 304.4625, Y 57.0565, Z -4.6667, A 0.000, B 0.000, C 0.000 }
gfCNCPoint3[25551] = {X 304.7761, Y 56.1603, Z -4.6667, A 0.000, B 0.000, C 0.000 }
gfCNCPoint3[25552] = {X 305.2813, Y 55.3564, Z -4.6667, A 0.000, B 0.000, C 0.000 }
gfCNCPoint3[25553] = {X 305.9526, Y 54.6850, Z -4.6667, A 0.000, B 0.000, C 0.000 }
gfCNCPoint3[25554] = {X 306.7566, Y 54.1799, Z -4.6667, A 0.000, B 0.000, C 0.000 }
gfCNCPoint3[25555] = {X 307.6527, Y 53.8663, Z -4.6667, A 0.000, B 0.000, C 0.000 }
gfCNCPoint3[25556] = {X 308.5962, Y 53.7600, Z -4.6667, A 0.000, B 0.000, C 0.000 }
gfCNCPoint3[25557] = {X 324.3107, Y 53.7600, Z -4.6667, A 0.000, B 0.000, C 0.000 }
gfCNCPoint3[25558] = {X 325.2542, Y 53.8663, Z -4.6667, A 0.000, B 0.000, C 0.000 }
gfCNCPoint3[25559] = {X 326.1504, Y 54.1799, Z -4.6667, A 0.000, B 0.000, C 0.000 }
gfCNCPoint3[25560] = {X 326.9543, Y 54.6850, Z -4.6667, A 0.000, B 0.000, C 0.000 }
gfCNCPoint3[25561] = {X 327.6257, Y 55.3564, Z -4.6667, A 0.000, B 0.000, C 0.000 }
gfCNCPoint3[25562] = {X 328.1308, Y 56.1603, Z -4.6667, A 0.000, B 0.000, C 0.000 }
gfCNCPoint3[25563] = {X 328.4444, Y 57.0565, Z -4.6667, A 0.000, B 0.000, C 0.000 }
gfCNCPoint3[25564] = {X 328.5507, Y 58.0000, Z -4.6667, A 0.000, B 0.000, C 0.000 }
gfCNCPoint3[25565] = {X 328.5507, Y 58.9355, Z -4.6667, A 0.000, B 0.000, C 0.000 }
gfCNCPoint3[25566] = {X 328.4562, Y 59.8053, Z -4.6667, A 0.000, B 0.000, C 0.000 }
gfCNCPoint3[25567] = {X 328.1868, Y 60.6377, Z -4.6667, A 0.000, B 0.000, C 0.000 }
gfCNCPoint3[25568] = {X 327.7537, Y 61.3979, Z -4.6667, A 0.000, B 0.000, C 0.000 }
gfCNCPoint3[25569] = {X 327.1750, Y 62.0541, Z -4.6667, A 0.000, B 0.000, C 0.000 }
gfCNCPoint3[25570] = {X 326.4750, Y 62.5789, Z -4.6667, A 0.000, B 0.000, C 0.000 }
gfCNCPoint3[25571] = {X 325.6827, Y 62.9503, Z -4.6667, A 0.000, B 0.000, C 0.000 }
gfCNCPoint3[25572] = {X 324.8316, Y 63.1528, Z -4.6667, A 0.000, B 0.000, C 0.000 }
gfCNCPoint3[25573] = {X 324.8332, Y 83.2300, Z -4.6667, A 0.000, B 0.000, C 0.000 }
gfCNCPoint3[25574] = {X 324.8468, Y 84.6150, Z -4.6667, A 0.000, B 0.000, C 0.000 }
gfCNCPoint3[25575] = {X 324.9257, Y 85.8671, Z -4.6667, A 0.000, B 0.000, C 0.000 }
gfCNCPoint3[25576] = {X 325.1520, Y 87.1012, Z -4.6667, A 0.000, B 0.000, C 0.000 }
gfCNCPoint3[25577] = {X 325.4128, Y 87.3910, Z -4.6667, A 0.000, B 0.000, C 0.000 }
gfCNCPoint3[25578] = {X 325.7358, Y 87.6093, Z -4.6667, A 0.000, B 0.000, C 0.000 }
gfCNCPoint3[25579] = {X 326.1875, Y 87.8647, Z -4.6667, A 0.000, B 0.000, C 0.000 }
gfCNCPoint3[25580] = {X 327.6346, Y 88.4654, Z -4.6667, A 0.000, B 0.000, C 0.000 }
gfCNCPoint3[25581] = {X 329.1388, Y 88.9039, Z -4.6667, A 0.000, B 0.000, C 0.000 }
gfCNCPoint3[25582] = {X 332.2203, Y 89.5209, Z -4.6667, A 0.000, B 0.000, C 0.000 }
gfCNCPoint3[25583] = {X 335.3382, Y 89.9146, Z -4.6667, A 0.000, B 0.000, C 0.000 }
gfCNCPoint3[25584] = {X 339.4789, Y 90.2347, Z -4.6667, A 0.000, B 0.000, C 0.000 }
gfCNCPoint3[25585] = {X 343.6280, Y 90.4144, Z -4.6667, A 0.000, B 0.000, C 0.000 }
gfCNCPoint3[25586] = {X 347.7809, Y 90.4534, Z -4.6667, A 0.000, B 0.000, C 0.000 }
gfCNCPoint3[25587] = {X 352.1650, Y 90.4149, Z -4.6667, A 0.000, B 0.000, C 0.000 }
gfCNCPoint3[25588] = {X 356.5449, Y 90.2189, Z -4.6667, A 0.000, B 0.000, C 0.000 }
gfCNCPoint3[25589] = {X 360.9150, Y 89.8657, Z -4.6667, A 0.000, B 0.000, C 0.000 }
gfCNCPoint3[25590] = {X 363.2338, Y 89.5773, Z -4.6667, A 0.000, B 0.000, C 0.000 }
gfCNCPoint3[25591] = {X 365.5310, Y 89.1500, Z -4.6667, A 0.000, B 0.000, C 0.000 }
gfCNCPoint3[25592] = {X 367.7985, Y 88.5855, Z -4.6667, A 0.000, B 0.000, C 0.000 }
gfCNCPoint3[25593] = {X 368.7387, Y 88.2694, Z -4.6667, A 0.000, B 0.000, C 0.000 }
gfCNCPoint3[25594] = {X 369.6376, Y 87.8498, Z -4.6667, A 0.000, B 0.000, C 0.000 }
gfCNCPoint3[25595] = {X 370.4838, Y 87.3321, Z -4.6667, A 0.000, B 0.000, C 0.000 }
gfCNCPoint3[25596] = {X 370.6556, Y 87.1533, Z -4.6667, A 0.000, B 0.000, C 0.000 }
gfCNCPoint3[25597] = {X 370.7441, Y 86.9218, Z -4.6667, A 0.000, B 0.000, C 0.000 }
gfCNCPoint3[25598] = {X 370.9360, Y 85.3803, Z -4.6667, A 0.000, B 0.000, C 0.000 }
gfCNCPoint3[25599] = {X 371.0001, Y 83.8283, Z -4.6667, A 0.000, B 0.000, C 0.000 }
gfCNCPoint3[25600] = {X 371.0005, Y 63.1422, Z -4.6667, A 0.000, B 0.000, C 0.000 }
gfCNCPoint3[25601] = {X 370.1519, Y 62.9475, Z -4.6667, A 0.000, B 0.000, C 0.000 }
gfCNCPoint3[25602] = {X 369.3610, Y 62.5836, Z -4.6667, A 0.000, B 0.000, C 0.000 }
gfCNCPoint3[25603] = {X 368.6611, Y 62.0659, Z -4.6667, A 0.000, B 0.000, C 0.000 }
gfCNCPoint3[25604] = {X 368.0817, Y 61.4161, Z -4.6667, A 0.000, B 0.000, C 0.000 }
gfCNCPoint3[25605] = {X 367.6472, Y 60.6616, Z -4.6667, A 0.000, B 0.000, C 0.000 }
gfCNCPoint3[25606] = {X 367.3760, Y 59.8343, Z -4.6667, A 0.000, B 0.000, C 0.000 }
gfCNCPoint3[25607] = {X 367.2794, Y 58.9691, Z -4.6667, A 0.000, B 0.000, C 0.000 }
gfCNCPoint3[25608] = {X 367.2793, Y 58.0000, Z -4.6667, A 0.000, B 0.000, C 0.000 }
gfCNCPoint3[25609] = {X 367.3856, Y 57.0565, Z -4.6667, A 0.000, B 0.000, C 0.000 }
gfCNCPoint3[25610] = {X 367.6992, Y 56.1603, Z -4.6667, A 0.000, B 0.000, C 0.000 }
gfCNCPoint3[25611] = {X 368.2043, Y 55.3564, Z -4.6667, A 0.000, B 0.000, C 0.000 }
gfCNCPoint3[25612] = {X 368.8757, Y 54.6850, Z -4.6667, A 0.000, B 0.000, C 0.000 }
gfCNCPoint3[25613] = {X 369.6796, Y 54.1799, Z -4.6667, A 0.000, B 0.000, C 0.000 }
gfCNCPoint3[25614] = {X 370.5758, Y 53.8663, Z -4.6667, A 0.000, B 0.000, C 0.000 }
gfCNCPoint3[25615] = {X 371.5193, Y 53.7600, Z -4.6667, A 0.000, B 0.000, C 0.000 }
gfCNCPoint3[25616] = {X 388.0597, Y 53.7600, Z -4.6667, A 0.000, B 0.000, C 0.000 }
gfCNCPoint3[25617] = {X 389.0032, Y 53.8663, Z -4.6667, A 0.000, B 0.000, C 0.000 }
gfCNCPoint3[25618] = {X 389.8993, Y 54.1799, Z -4.6667, A 0.000, B 0.000, C 0.000 }
gfCNCPoint3[25619] = {X 390.7033, Y 54.6850, Z -4.6667, A 0.000, B 0.000, C 0.000 }
gfCNCPoint3[25620] = {X 391.3746, Y 55.3564, Z -4.6667, A 0.000, B 0.000, C 0.000 }
gfCNCPoint3[25621] = {X 391.8798, Y 56.1603, Z -4.6667, A 0.000, B 0.000, C 0.000 }
gfCNCPoint3[25622] = {X 392.1934, Y 57.0565, Z -4.6667, A 0.000, B 0.000, C 0.000 }
gfCNCPoint3[25623] = {X 392.2997, Y 58.0000, Z -4.6667, A 0.000, B 0.000, C 0.000 }
gfCNCPoint3[25624] = {X 392.2997, Y 58.9342, Z -4.6667, A 0.000, B 0.000, C 0.000 }
gfCNCPoint3[25625] = {X 392.1881, Y 59.9005, Z -4.6667, A 0.000, B 0.000, C 0.000 }
gfCNCPoint3[25626] = {X 391.8592, Y 60.8160, Z -4.6667, A 0.000, B 0.000, C 0.000 }
gfCNCPoint3[25627] = {X 391.4159, Y 61.5272, Z -4.6667, A 0.000, B 0.000, C 0.000 }
gfCNCPoint3[25628] = {X 390.8422, Y 62.1379, Z -4.6667, A 0.000, B 0.000, C 0.000 }
gfCNCPoint3[25629] = {X 390.1599, Y 62.6246, Z -4.6667, A 0.000, B 0.000, C 0.000 }
gfCNCPoint3[25630] = {X 389.3957, Y 62.9684, Z -4.6667, A 0.000, B 0.000, C 0.000 }
gfCNCPoint3[25631] = {X 388.5790, Y 63.1560, Z -4.6667, A 0.000, B 0.000, C 0.000 }
gfCNCPoint3[25632] = {X 388.5769, Y 84.6150, Z -4.6667, A 0.000, B 0.000, C 0.000 }
gfCNCPoint3[25633] = {X 388.5173, Y 86.2665, Z -4.6667, A 0.000, B 0.000, C 0.000 }
gfCNCPoint3[25634] = {X 388.3138, Y 87.9065, Z -4.6667, A 0.000, B 0.000, C 0.000 }
gfCNCPoint3[25635] = {X 387.9681, Y 89.5224, Z -4.6667, A 0.000, B 0.000, C 0.000 }
gfCNCPoint3[25636] = {X 387.4395, Y 91.0991, Z -4.6667, A 0.000, B 0.000, C 0.000 }
gfCNCPoint3[25637] = {X 386.6949, Y 92.5860, Z -4.6667, A 0.000, B 0.000, C 0.000 }
gfCNCPoint3[25638] = {X 385.7492, Y 93.9538, Z -4.6667, A 0.000, B 0.000, C 0.000 }
gfCNCPoint3[25639] = {X 384.6210, Y 95.1755, Z -4.6667, A 0.000, B 0.000, C 0.000 }
gfCNCPoint3[25640] = {X 383.1131, Y 96.4461, Z -4.6667, A 0.000, B 0.000, C 0.000 }
gfCNCPoint3[25641] = {X 381.4788, Y 97.5494, Z -4.6667, A 0.000, B 0.000, C 0.000 }
gfCNCPoint3[25642] = {X 379.7367, Y 98.4730, Z -4.6667, A 0.000, B 0.000, C 0.000 }
gfCNCPoint3[25643] = {X 377.4708, Y 99.4269, Z -4.6667, A 0.000, B 0.000, C 0.000 }
gfCNCPoint3[25644] = {X 375.1421, Y 100.2153, Z -4.6667, A 0.000, B 0.000, C 0.000 }
gfCNCPoint3[25645] = {X 372.7628, Y 100.8342, Z -4.6667, A 0.000, B 0.000, C 0.000 }
gfCNCPoint3[25646] = {X 368.8561, Y 101.5875, Z -4.6667, A 0.000, B 0.000, C 0.000 }
gfCNCPoint3[25647] = {X 364.9169, Y 102.1472, Z -4.6667, A 0.000, B 0.000, C 0.000 }
gfCNCPoint3[25648] = {X 360.9550, Y 102.5120, Z -4.6667, A 0.000, B 0.000, C 0.000 }
gfCNCPoint3[25649] = {X 357.0996, Y 102.7368, Z -4.6667, A 0.000, B 0.000, C 0.000 }
gfCNCPoint3[25650] = {X 353.2405, Y 102.8821, Z -4.6667, A 0.000, B 0.000, C 0.000 }
gfCNCPoint3[25651] = {X 353.3497, Y 106.8806, Z -4.6667, A 0.000, B 0.000, C 0.000 }
gfCNCPoint3[25652] = {X 353.2383, Y 102.8021, Z -4.6667, A 0.000, B 0.000, C 0.000 }
gfCNCPoint3[25653] = {X 348.1838, Y 102.8719, Z -4.6667, A 0.000, B 0.000, C 0.000 }
gfCNCPoint3[25654] = {X 343.1292, Y 102.8052, Z -4.6667, A 0.000, B 0.000, C 0.000 }
gfCNCPoint3[25655] = {X 338.0783, Y 102.6020, Z -4.6667, A 0.000, B 0.000, C 0.000 }
gfCNCPoint3[25656] = {X 334.1305, Y 102.3256, Z -4.6667, A 0.000, B 0.000, C 0.000 }
gfCNCPoint3[25657] = {X 330.1977, Y 101.8844, Z -4.6667, A 0.000, B 0.000, C 0.000 }
gfCNCPoint3[25658] = {X 326.2868, Y 101.2794, Z -4.6667, A 0.000, B 0.000, C 0.000 }
gfCNCPoint3[25659] = {X 323.4483, Y 100.6780, Z -4.6667, A 0.000, B 0.000, C 0.000 }
gfCNCPoint3[25660] = {X 320.6620, Y 99.8682, Z -4.6667, A 0.000, B 0.000, C 0.000 }
gfCNCPoint3[25661] = {X 317.9433, Y 98.8547, Z -4.6667, A 0.000, B 0.000, C 0.000 }
gfCNCPoint3[25662] = {X 316.4429, Y 98.1617, Z -4.6667, A 0.000, B 0.000, C 0.000 }
gfCNCPoint3[25663] = {X 315.0055, Y 97.3462, Z -4.6667, A 0.000, B 0.000, C 0.000 }
gfCNCPoint3[25664] = {X 313.6409, Y 96.4139, Z -4.6667, A 0.000, B 0.000, C 0.000 }
gfCNCPoint3[25665] = {X 312.3587, Y 95.3712, Z -4.6667, A 0.000, B 0.000, C 0.000 }
gfCNCPoint3[25666] = {X 311.3684, Y 94.3862, Z -4.6667, A 0.000, B 0.000, C 0.000 }
gfCNCPoint3[25667] = {X 310.5019, Y 93.2906, Z -4.6667, A 0.000, B 0.000, C 0.000 }
gfCNCPoint3[25668] = {X 309.7713, Y 92.1001, Z -4.6667, A 0.000, B 0.000, C 0.000 }
gfCNCPoint3[25669] = {X 309.1872, Y 90.8313, Z -4.6667, A 0.000, B 0.000, C 0.000 }
gfCNCPoint3[25670] = {X 308.7575, Y 89.5022, Z -4.6667, A 0.000, B 0.000, C 0.000 }
gfCNCPoint3[25671] = {X 308.4169, Y 87.8925, Z -4.6667, A 0.000, B 0.000, C 0.000 }
gfCNCPoint3[25672] = {X 308.2157, Y 86.2595, Z -4.6667, A 0.000, B 0.000, C 0.000 }
gfCNCPoint3[25673] = {X 308.1554, Y 84.6152, Z -4.6667, A 0.000, B 0.000, C 0.000 }
gfCNCPoint3[25674] = {X 308.1566, Y 63.0708, Z -4.6667, A 0.000, B 0.000, C 0.000 }
gfCNCPoint3[25675] = {X 307.3115, Y 62.8907, Z -4.6667, A 0.000, B 0.000, C 0.000 }
gfCNCPoint3[25676] = {X 306.5218, Y 62.5399, Z -4.6667, A 0.000, B 0.000, C 0.000 }
gfCNCPoint3[25677] = {X 305.8216, Y 62.0336, Z -4.6667, A 0.000, B 0.000, C 0.000 }
gfCNCPoint3[25678] = {X 305.2411, Y 61.3935, Z -4.6667, A 0.000, B 0.000, C 0.000 }
gfCNCPoint3[25679] = {X 304.8054, Y 60.6472, Z -4.6667, A 0.000, B 0.000, C 0.000 }
gfCNCPoint3[25680] = {X 304.5332, Y 59.8271, Z -4.6667, A 0.000, B 0.000, C 0.000 }
gfCNCPoint3[25681] = {X 304.4364, Y 58.9684, Z -4.6667, A 0.000, B 0.000, C 0.000 }
gfCNCPoint3[25682] = {X 304.4362, Y 58.0000, Z -4.6667, A 0.000, B 0.000, C 0.000 }
gfCNCPoint3[25683] = {X 304.5405, Y 57.0743, Z -4.6667, A 0.000, B 0.000, C 0.000 }
gfCNCPoint3[25684] = {X 304.8482, Y 56.1950, Z -4.6667, A 0.000, B 0.000, C 0.000 }
gfCNCPoint3[25685] = {X 305.3438, Y 55.4063, Z -4.6667, A 0.000, B 0.000, C 0.000 }
gfCNCPoint3[25686] = {X 306.0025, Y 54.7476, Z -4.6667, A 0.000, B 0.000, C 0.000 }
gfCNCPoint3[25687] = {X 306.7913, Y 54.2520, Z -4.6667, A 0.000, B 0.000, C 0.000 }
gfCNCPoint3[25688] = {X 307.6705, Y 53.9443, Z -4.6667, A 0.000, B 0.000, C 0.000 }
gfCNCPoint3[25689] = {X 308.5962, Y 53.8400, Z -4.6667, A 0.000, B 0.000, C 0.000 }
gfCNCPoint3[25690] = {X 324.3107, Y 53.8400, Z -4.6667, A 0.000, B 0.000, C 0.000 }
gfCNCPoint3[25691] = {X 325.2364, Y 53.9443, Z -4.6667, A 0.000, B 0.000, C 0.000 }
gfCNCPoint3[25692] = {X 326.1156, Y 54.2520, Z -4.6667, A 0.000, B 0.000, C 0.000 }
gfCNCPoint3[25693] = {X 326.9044, Y 54.7476, Z -4.6667, A 0.000, B 0.000, C 0.000 }
gfCNCPoint3[25694] = {X 327.5631, Y 55.4063, Z -4.6667, A 0.000, B 0.000, C 0.000 }
gfCNCPoint3[25695] = {X 328.0587, Y 56.1950, Z -4.6667, A 0.000, B 0.000, C 0.000 }
gfCNCPoint3[25696] = {X 328.3664, Y 57.0743, Z -4.6667, A 0.000, B 0.000, C 0.000 }
gfCNCPoint3[25697] = {X 328.4707, Y 58.0000, Z -4.6667, A 0.000, B 0.000, C 0.000 }
gfCNCPoint3[25698] = {X 328.4707, Y 58.9350, Z -4.6667, A 0.000, B 0.000, C 0.000 }
gfCNCPoint3[25699] = {X 328.3759, Y 59.7984, Z -4.6667, A 0.000, B 0.000, C 0.000 }
gfCNCPoint3[25700] = {X 328.1055, Y 60.6237, Z -4.6667, A 0.000, B 0.000, C 0.000 }
gfCNCPoint3[25701] = {X 327.6711, Y 61.3758, Z -4.6667, A 0.000, B 0.000, C 0.000 }
gfCNCPoint3[25702] = {X 327.0912, Y 62.0224, Z -4.6667, A 0.000, B 0.000, C 0.000 }
gfCNCPoint3[25703] = {X 326.3907, Y 62.5358, Z -4.6667, A 0.000, B 0.000, C 0.000 }
gfCNCPoint3[25704] = {X 325.5995, Y 62.8942, Z -4.6667, A 0.000, B 0.000, C 0.000 }
gfCNCPoint3[25705] = {X 324.7516, Y 63.0820, Z -4.6667, A 0.000, B 0.000, C 0.000 }
gfCNCPoint3[25706] = {X 324.7532, Y 83.2304, Z -4.6667, A 0.000, B 0.000, C 0.000 }
gfCNCPoint3[25707] = {X 324.7668, Y 84.6153, Z -4.6667, A 0.000, B 0.000, C 0.000 }
gfCNCPoint3[25708] = {X 324.8472, Y 85.8842, Z -4.6667, A 0.000, B 0.000, C 0.000 }
gfCNCPoint3[25709] = {X 325.0779, Y 87.1346, Z -4.6667, A 0.000, B 0.000, C 0.000 }
gfCNCPoint3[25710] = {X 325.3539, Y 87.4458, Z -4.6667, A 0.000, B 0.000, C 0.000 }
gfCNCPoint3[25711] = {X 325.6979, Y 87.6798, Z -4.6667, A 0.000, B 0.000, C 0.000 }
gfCNCPoint3[25712] = {X 326.1504, Y 87.9356, Z -4.6667, A 0.000, B 0.000, C 0.000 }
gfCNCPoint3[25713] = {X 327.6068, Y 88.5404, Z -4.6667, A 0.000, B 0.000, C 0.000 }
gfCNCPoint3[25714] = {X 329.1206, Y 88.9818, Z -4.6667, A 0.000, B 0.000, C 0.000 }
gfCNCPoint3[25715] = {X 332.2076, Y 89.5999, Z -4.6667, A 0.000, B 0.000, C 0.000 }
gfCNCPoint3[25716] = {X 335.3310, Y 89.9942, Z -4.6667, A 0.000, B 0.000, C 0.000 }
gfCNCPoint3[25717] = {X 339.4743, Y 90.3146, Z -4.6667, A 0.000, B 0.000, C 0.000 }
gfCNCPoint3[25718] = {X 343.6261, Y 90.4944, Z -4.6667, A 0.000, B 0.000, C 0.000 }
gfCNCPoint3[25719] = {X 347.7815, Y 90.5334, Z -4.6667, A 0.000, B 0.000, C 0.000 }
gfCNCPoint3[25720] = {X 352.1681, Y 90.4949, Z -4.6667, A 0.000, B 0.000, C 0.000 }
gfCNCPoint3[25721] = {X 356.5504, Y 90.2987, Z -4.6667, A 0.000, B 0.000, C 0.000 }
gfCNCPoint3[25722] = {X 360.9228, Y 89.9453, Z -4.6667, A 0.000, B 0.000, C 0.000 }
gfCNCPoint3[25723] = {X 363.2463, Y 89.6563, Z -4.6667, A 0.000, B 0.000, C 0.000 }
gfCNCPoint3[25724] = {X 365.5481, Y 89.2282, Z -4.6667, A 0.000, B 0.000, C 0.000 }
gfCNCPoint3[25725] = {X 367.8201, Y 88.6625, Z -4.6667, A 0.000, B 0.000, C 0.000 }
gfCNCPoint3[25726] = {X 368.7687, Y 88.3435, Z -4.6667, A 0.000, B 0.000, C 0.000 }
gfCNCPoint3[25727] = {X 369.6756, Y 87.9202, Z -4.6667, A 0.000, B 0.000, C 0.000 }
gfCNCPoint3[25728] = {X 370.5293, Y 87.3979, Z -4.6667, A 0.000, B 0.000, C 0.000 }
gfCNCPoint3[25729] = {X 370.7231, Y 87.1962, Z -4.6667, A 0.000, B 0.000, C 0.000 }
gfCNCPoint3[25730] = {X 370.8230, Y 86.9349, Z -4.6667, A 0.000, B 0.000, C 0.000 }
gfCNCPoint3[25731] = {X 371.0158, Y 85.3869, Z -4.6667, A 0.000, B 0.000, C 0.000 }
gfCNCPoint3[25732] = {X 371.0801, Y 83.8283, Z -4.6667, A 0.000, B 0.000, C 0.000 }
gfCNCPoint3[25733] = {X 371.0805, Y 63.0709, Z -4.6667, A 0.000, B 0.000, C 0.000 }
gfCNCPoint3[25734] = {X 370.9780, Y 63.0587, Z -4.6667, A 0.000, B 0.000, C 0.000 }
gfCNCPoint3[25735] = {X 370.8758, Y 63.0440, Z -4.6667, A 0.000, B 0.000, C 0.000 }
gfCNCPoint3[25736] = {X 369.9383, Y 62.7819, Z -4.6667, A 0.000, B 0.000, C 0.000 }
gfCNCPoint3[25737] = {X 369.0873, Y 62.3092, Z -4.6667, A 0.000, B 0.000, C 0.000 }
gfCNCPoint3[25738] = {X 368.3696, Y 61.6516, Z -4.6667, A 0.000, B 0.000, C 0.000 }
gfCNCPoint3[25739] = {X 367.8243, Y 60.8452, Z -4.6667, A 0.000, B 0.000, C 0.000 }
gfCNCPoint3[25740] = {X 367.4813, Y 59.9342, Z -4.6667, A 0.000, B 0.000, C 0.000 }
gfCNCPoint3[25741] = {X 367.3594, Y 58.9684, Z -4.6667, A 0.000, B 0.000, C 0.000 }
gfCNCPoint3[25742] = {X 367.3593, Y 58.0000, Z -4.6667, A 0.000, B 0.000, C 0.000 }
gfCNCPoint3[25743] = {X 367.4636, Y 57.0743, Z -4.6667, A 0.000, B 0.000, C 0.000 }
gfCNCPoint3[25744] = {X 367.7713, Y 56.1950, Z -4.6667, A 0.000, B 0.000, C 0.000 }
gfCNCPoint3[25745] = {X 368.2669, Y 55.4063, Z -4.6667, A 0.000, B 0.000, C 0.000 }
gfCNCPoint3[25746] = {X 368.9256, Y 54.7476, Z -4.6667, A 0.000, B 0.000, C 0.000 }
gfCNCPoint3[25747] = {X 369.7143, Y 54.2520, Z -4.6667, A 0.000, B 0.000, C 0.000 }
gfCNCPoint3[25748] = {X 370.5936, Y 53.9443, Z -4.6667, A 0.000, B 0.000, C 0.000 }
gfCNCPoint3[25749] = {X 371.5193, Y 53.8400, Z -4.6667, A 0.000, B 0.000, C 0.000 }
gfCNCPoint3[25750] = {X 388.0597, Y 53.8400, Z -4.6667, A 0.000, B 0.000, C 0.000 }
gfCNCPoint3[25751] = {X 388.9854, Y 53.9443, Z -4.6667, A 0.000, B 0.000, C 0.000 }
gfCNCPoint3[25752] = {X 389.8646, Y 54.2520, Z -4.6667, A 0.000, B 0.000, C 0.000 }
gfCNCPoint3[25753] = {X 390.6534, Y 54.7476, Z -4.6667, A 0.000, B 0.000, C 0.000 }
gfCNCPoint3[25754] = {X 391.3121, Y 55.4063, Z -4.6667, A 0.000, B 0.000, C 0.000 }
gfCNCPoint3[25755] = {X 391.8077, Y 56.1950, Z -4.6667, A 0.000, B 0.000, C 0.000 }
gfCNCPoint3[25756] = {X 392.1154, Y 57.0743, Z -4.6667, A 0.000, B 0.000, C 0.000 }
gfCNCPoint3[25757] = {X 392.2197, Y 58.0000, Z -4.6667, A 0.000, B 0.000, C 0.000 }
gfCNCPoint3[25758] = {X 392.2197, Y 58.9342, Z -4.6667, A 0.000, B 0.000, C 0.000 }
gfCNCPoint3[25759] = {X 392.1102, Y 59.8823, Z -4.6667, A 0.000, B 0.000, C 0.000 }
gfCNCPoint3[25760] = {X 391.7875, Y 60.7805, Z -4.6667, A 0.000, B 0.000, C 0.000 }
gfCNCPoint3[25761] = {X 391.2441, Y 61.6118, Z -4.6667, A 0.000, B 0.000, C 0.000 }
gfCNCPoint3[25762] = {X 390.5200, Y 62.2916, Z -4.6667, A 0.000, B 0.000, C 0.000 }
gfCNCPoint3[25763] = {X 389.6561, Y 62.7815, Z -4.6667, A 0.000, B 0.000, C 0.000 }
gfCNCPoint3[25764] = {X 388.7010, Y 63.0538, Z -4.6667, A 0.000, B 0.000, C 0.000 }
gfCNCPoint3[25765] = {X 388.6008, Y 63.0686, Z -4.6667, A 0.000, B 0.000, C 0.000 }
gfCNCPoint3[25766] = {X 388.5002, Y 63.0810, Z -4.6667, A 0.000, B 0.000, C 0.000 }
gfCNCPoint3[25767] = {X 388.4969, Y 84.6154, Z -4.6667, A 0.000, B 0.000, C 0.000 }
gfCNCPoint3[25768] = {X 388.4376, Y 86.2599, Z -4.6667, A 0.000, B 0.000, C 0.000 }
gfCNCPoint3[25769] = {X 388.2349, Y 87.8931, Z -4.6667, A 0.000, B 0.000, C 0.000 }
gfCNCPoint3[25770] = {X 387.8906, Y 89.5023, Z -4.6667, A 0.000, B 0.000, C 0.000 }
gfCNCPoint3[25771] = {X 387.3656, Y 91.0683, Z -4.6667, A 0.000, B 0.000, C 0.000 }
gfCNCPoint3[25772] = {X 386.6261, Y 92.5452, Z -4.6667, A 0.000, B 0.000, C 0.000 }
gfCNCPoint3[25773] = {X 385.6868, Y 93.9038, Z -4.6667, A 0.000, B 0.000, C 0.000 }
gfCNCPoint3[25774] = {X 384.5662, Y 95.1172, Z -4.6667, A 0.000, B 0.000, C 0.000 }
gfCNCPoint3[25775] = {X 383.0648, Y 96.3823, Z -4.6667, A 0.000, B 0.000, C 0.000 }
gfCNCPoint3[25776] = {X 381.4376, Y 97.4808, Z -4.6667, A 0.000, B 0.000, C 0.000 }
gfCNCPoint3[25777] = {X 379.7030, Y 98.4004, Z -4.6667, A 0.000, B 0.000, C 0.000 }
gfCNCPoint3[25778] = {X 377.4424, Y 99.3521, Z -4.6667, A 0.000, B 0.000, C 0.000 }
gfCNCPoint3[25779] = {X 375.1192, Y 100.1387, Z -4.6667, A 0.000, B 0.000, C 0.000 }
gfCNCPoint3[25780] = {X 372.7455, Y 100.7561, Z -4.6667, A 0.000, B 0.000, C 0.000 }
gfCNCPoint3[25781] = {X 368.8427, Y 101.5086, Z -4.6667, A 0.000, B 0.000, C 0.000 }
gfCNCPoint3[25782] = {X 364.9075, Y 102.0678, Z -4.6667, A 0.000, B 0.000, C 0.000 }
gfCNCPoint3[25783] = {X 360.9496, Y 102.4322, Z -4.6667, A 0.000, B 0.000, C 0.000 }
gfCNCPoint3[25784] = {X 357.0958, Y 102.6569, Z -4.6667, A 0.000, B 0.000, C 0.000 }
gfCNCPoint3[25785] = {X 353.2383, Y 102.8021, Z -4.6667, A 0.000, B 0.000, C 0.000 }
gfCNCPoint3[25786] = {X 353.3476, Y 106.8006, Z -4.6667, A 0.000, B 0.000, C 0.000 }
gfCNCPoint3[25787] = {X 353.2361, Y 102.7222, Z -4.6667, A 0.000, B 0.000, C 0.000 }
gfCNCPoint3[25788] = {X 348.1837, Y 102.7919, Z -4.6667, A 0.000, B 0.000, C 0.000 }
gfCNCPoint3[25789] = {X 343.1313, Y 102.7252, Z -4.6667, A 0.000, B 0.000, C 0.000 }
gfCNCPoint3[25790] = {X 338.0825, Y 102.5221, Z -4.6667, A 0.000, B 0.000, C 0.000 }
gfCNCPoint3[25791] = {X 334.1379, Y 102.2459, Z -4.6667, A 0.000, B 0.000, C 0.000 }
gfCNCPoint3[25792] = {X 330.2084, Y 101.8051, Z -4.6667, A 0.000, B 0.000, C 0.000 }
gfCNCPoint3[25793] = {X 326.3006, Y 101.2006, Z -4.6667, A 0.000, B 0.000, C 0.000 }
gfCNCPoint3[25794] = {X 323.4678, Y 100.6004, Z -4.6667, A 0.000, B 0.000, C 0.000 }
gfCNCPoint3[25795] = {X 320.6872, Y 99.7923, Z -4.6667, A 0.000, B 0.000, C 0.000 }
gfCNCPoint3[25796] = {X 317.9739, Y 98.7808, Z -4.6667, A 0.000, B 0.000, C 0.000 }
gfCNCPoint3[25797] = {X 316.4796, Y 98.0906, Z -4.6667, A 0.000, B 0.000, C 0.000 }
gfCNCPoint3[25798] = {X 315.0479, Y 97.2784, Z -4.6667, A 0.000, B 0.000, C 0.000 }
gfCNCPoint3[25799] = {X 313.6888, Y 96.3498, Z -4.6667, A 0.000, B 0.000, C 0.000 }
gfCNCPoint3[25800] = {X 312.4117, Y 95.3113, Z -4.6667, A 0.000, B 0.000, C 0.000 }
gfCNCPoint3[25801] = {X 311.4281, Y 94.3330, Z -4.6667, A 0.000, B 0.000, C 0.000 }
gfCNCPoint3[25802] = {X 310.5675, Y 93.2449, Z -4.6667, A 0.000, B 0.000, C 0.000 }
gfCNCPoint3[25803] = {X 309.8419, Y 92.0624, Z -4.6667, A 0.000, B 0.000, C 0.000 }
gfCNCPoint3[25804] = {X 309.2617, Y 90.8022, Z -4.6667, A 0.000, B 0.000, C 0.000 }
gfCNCPoint3[25805] = {X 308.8350, Y 89.4822, Z -4.6667, A 0.000, B 0.000, C 0.000 }
gfCNCPoint3[25806] = {X 308.4958, Y 87.8792, Z -4.6667, A 0.000, B 0.000, C 0.000 }
gfCNCPoint3[25807] = {X 308.2955, Y 86.2530, Z -4.6667, A 0.000, B 0.000, C 0.000 }
gfCNCPoint3[25808] = {X 308.2354, Y 84.6156, Z -4.6667, A 0.000, B 0.000, C 0.000 }
gfCNCPoint3[25809] = {X 308.2366, Y 62.9982, Z -4.6667, A 0.000, B 0.000, C 0.000 }
gfCNCPoint3[25810] = {X 307.3949, Y 62.8332, Z -4.6667, A 0.000, B 0.000, C 0.000 }
gfCNCPoint3[25811] = {X 306.6063, Y 62.4959, Z -4.6667, A 0.000, B 0.000, C 0.000 }
gfCNCPoint3[25812] = {X 305.9057, Y 62.0012, Z -4.6667, A 0.000, B 0.000, C 0.000 }
gfCNCPoint3[25813] = {X 305.3239, Y 61.3709, Z -4.6667, A 0.000, B 0.000, C 0.000 }
gfCNCPoint3[25814] = {X 304.8868, Y 60.6330, Z -4.6667, A 0.000, B 0.000, C 0.000 }
gfCNCPoint3[25815] = {X 304.6136, Y 59.8199, Z -4.6667, A 0.000, B 0.000, C 0.000 }
gfCNCPoint3[25816] = {X 304.5164, Y 58.9678, Z -4.6667, A 0.000, B 0.000, C 0.000 }
gfCNCPoint3[25817] = {X 304.5162, Y 58.0000, Z -4.6667, A 0.000, B 0.000, C 0.000 }
gfCNCPoint3[25818] = {X 304.6185, Y 57.0921, Z -4.6667, A 0.000, B 0.000, C 0.000 }
gfCNCPoint3[25819] = {X 304.9203, Y 56.2298, Z -4.6667, A 0.000, B 0.000, C 0.000 }
gfCNCPoint3[25820] = {X 305.4064, Y 55.4562, Z -4.6667, A 0.000, B 0.000, C 0.000 }
gfCNCPoint3[25821] = {X 306.0524, Y 54.8101, Z -4.6667, A 0.000, B 0.000, C 0.000 }
gfCNCPoint3[25822] = {X 306.8260, Y 54.3240, Z -4.6667, A 0.000, B 0.000, C 0.000 }
gfCNCPoint3[25823] = {X 307.6883, Y 54.0223, Z -4.6667, A 0.000, B 0.000, C 0.000 }
gfCNCPoint3[25824] = {X 308.5962, Y 53.9200, Z -4.6667, A 0.000, B 0.000, C 0.000 }
gfCNCPoint3[25825] = {X 324.3107, Y 53.9200, Z -4.6667, A 0.000, B 0.000, C 0.000 }
gfCNCPoint3[25826] = {X 325.2186, Y 54.0223, Z -4.6667, A 0.000, B 0.000, C 0.000 }
gfCNCPoint3[25827] = {X 326.0809, Y 54.3240, Z -4.6667, A 0.000, B 0.000, C 0.000 }
gfCNCPoint3[25828] = {X 326.8545, Y 54.8101, Z -4.6667, A 0.000, B 0.000, C 0.000 }
gfCNCPoint3[25829] = {X 327.5006, Y 55.4562, Z -4.6667, A 0.000, B 0.000, C 0.000 }
gfCNCPoint3[25830] = {X 327.9866, Y 56.2298, Z -4.6667, A 0.000, B 0.000, C 0.000 }
gfCNCPoint3[25831] = {X 328.2884, Y 57.0921, Z -4.6667, A 0.000, B 0.000, C 0.000 }
gfCNCPoint3[25832] = {X 328.3907, Y 58.0000, Z -4.6667, A 0.000, B 0.000, C 0.000 }
gfCNCPoint3[25833] = {X 328.3907, Y 58.9346, Z -4.6667, A 0.000, B 0.000, C 0.000 }
gfCNCPoint3[25834] = {X 328.2956, Y 59.7914, Z -4.6667, A 0.000, B 0.000, C 0.000 }
gfCNCPoint3[25835] = {X 328.0241, Y 60.6097, Z -4.6667, A 0.000, B 0.000, C 0.000 }
gfCNCPoint3[25836] = {X 327.5883, Y 61.3535, Z -4.6667, A 0.000, B 0.000, C 0.000 }
gfCNCPoint3[25837] = {X 327.0072, Y 61.9903, Z -4.6667, A 0.000, B 0.000, C 0.000 }
gfCNCPoint3[25838] = {X 326.3062, Y 62.4922, Z -4.6667, A 0.000, B 0.000, C 0.000 }
gfCNCPoint3[25839] = {X 325.5161, Y 62.8371, Z -4.6667, A 0.000, B 0.000, C 0.000 }
gfCNCPoint3[25840] = {X 324.6715, Y 63.0101, Z -4.6667, A 0.000, B 0.000, C 0.000 }
gfCNCPoint3[25841] = {X 324.6732, Y 83.2309, Z -4.6667, A 0.000, B 0.000, C 0.000 }
gfCNCPoint3[25842] = {X 324.6868, Y 84.6156, Z -4.6667, A 0.000, B 0.000, C 0.000 }
gfCNCPoint3[25843] = {X 324.7687, Y 85.9012, Z -4.6667, A 0.000, B 0.000, C 0.000 }
gfCNCPoint3[25844] = {X 325.0037, Y 87.1678, Z -4.6667, A 0.000, B 0.000, C 0.000 }
gfCNCPoint3[25845] = {X 325.2950, Y 87.5005, Z -4.6667, A 0.000, B 0.000, C 0.000 }
gfCNCPoint3[25846] = {X 325.6599, Y 87.7502, Z -4.6667, A 0.000, B 0.000, C 0.000 }
gfCNCPoint3[25847] = {X 326.1134, Y 88.0066, Z -4.6667, A 0.000, B 0.000, C 0.000 }
gfCNCPoint3[25848] = {X 327.5789, Y 88.6154, Z -4.6667, A 0.000, B 0.000, C 0.000 }
gfCNCPoint3[25849] = {X 329.1025, Y 89.0598, Z -4.6667, A 0.000, B 0.000, C 0.000 }
gfCNCPoint3[25850] = {X 332.1949, Y 89.6788, Z -4.6667, A 0.000, B 0.000, C 0.000 }
gfCNCPoint3[25851] = {X 335.3238, Y 90.0739, Z -4.6667, A 0.000, B 0.000, C 0.000 }
gfCNCPoint3[25852] = {X 339.4695, Y 90.3945, Z -4.6667, A 0.000, B 0.000, C 0.000 }
gfCNCPoint3[25853] = {X 343.6236, Y 90.5744, Z -4.6667, A 0.000, B 0.000, C 0.000 }
gfCNCPoint3[25854] = {X 347.7815, Y 90.6134, Z -4.6667, A 0.000, B 0.000, C 0.000 }
gfCNCPoint3[25855] = {X 352.1707, Y 90.5748, Z -4.6667, A 0.000, B 0.000, C 0.000 }
gfCNCPoint3[25856] = {X 356.5556, Y 90.3786, Z -4.6667, A 0.000, B 0.000, C 0.000 }
gfCNCPoint3[25857] = {X 360.9307, Y 90.0249, Z -4.6667, A 0.000, B 0.000, C 0.000 }
gfCNCPoint3[25858] = {X 363.2588, Y 89.7353, Z -4.6667, A 0.000, B 0.000, C 0.000 }
gfCNCPoint3[25859] = {X 365.5653, Y 89.3063, Z -4.6667, A 0.000, B 0.000, C 0.000 }
gfCNCPoint3[25860] = {X 367.8418, Y 88.7395, Z -4.6667, A 0.000, B 0.000, C 0.000 }
gfCNCPoint3[25861] = {X 368.7987, Y 88.4177, Z -4.6667, A 0.000, B 0.000, C 0.000 }
gfCNCPoint3[25862] = {X 369.7136, Y 87.9906, Z -4.6667, A 0.000, B 0.000, C 0.000 }
gfCNCPoint3[25863] = {X 370.5748, Y 87.4637, Z -4.6667, A 0.000, B 0.000, C 0.000 }
gfCNCPoint3[25864] = {X 370.7907, Y 87.2391, Z -4.6667, A 0.000, B 0.000, C 0.000 }
gfCNCPoint3[25865] = {X 370.9020, Y 86.9481, Z -4.6667, A 0.000, B 0.000, C 0.000 }
gfCNCPoint3[25866] = {X 371.0955, Y 85.3935, Z -4.6667, A 0.000, B 0.000, C 0.000 }
gfCNCPoint3[25867] = {X 371.1601, Y 83.8283, Z -4.6667, A 0.000, B 0.000, C 0.000 }
gfCNCPoint3[25868] = {X 371.1605, Y 62.9983, Z -4.6667, A 0.000, B 0.000, C 0.000 }
gfCNCPoint3[25869] = {X 371.0240, Y 62.9839, Z -4.6667, A 0.000, B 0.000, C 0.000 }
gfCNCPoint3[25870] = {X 370.8881, Y 62.9650, Z -4.6667, A 0.000, B 0.000, C 0.000 }
gfCNCPoint3[25871] = {X 369.9687, Y 62.7079, Z -4.6667, A 0.000, B 0.000, C 0.000 }
gfCNCPoint3[25872] = {X 369.1341, Y 62.2443, Z -4.6667, A 0.000, B 0.000, C 0.000 }
gfCNCPoint3[25873] = {X 368.4301, Y 61.5993, Z -4.6667, A 0.000, B 0.000, C 0.000 }
gfCNCPoint3[25874] = {X 367.8953, Y 60.8085, Z -4.6667, A 0.000, B 0.000, C 0.000 }
gfCNCPoint3[25875] = {X 367.5590, Y 59.9150, Z -4.6667, A 0.000, B 0.000, C 0.000 }
gfCNCPoint3[25876] = {X 367.4394, Y 58.9678, Z -4.6667, A 0.000, B 0.000, C 0.000 }
gfCNCPoint3[25877] = {X 367.4393, Y 58.0000, Z -4.6667, A 0.000, B 0.000, C 0.000 }
gfCNCPoint3[25878] = {X 367.5416, Y 57.0921, Z -4.6667, A 0.000, B 0.000, C 0.000 }
gfCNCPoint3[25879] = {X 367.8433, Y 56.2298, Z -4.6667, A 0.000, B 0.000, C 0.000 }
gfCNCPoint3[25880] = {X 368.3294, Y 55.4562, Z -4.6667, A 0.000, B 0.000, C 0.000 }
gfCNCPoint3[25881] = {X 368.9754, Y 54.8101, Z -4.6667, A 0.000, B 0.000, C 0.000 }
gfCNCPoint3[25882] = {X 369.7490, Y 54.3240, Z -4.6667, A 0.000, B 0.000, C 0.000 }
gfCNCPoint3[25883] = {X 370.6114, Y 54.0223, Z -4.6667, A 0.000, B 0.000, C 0.000 }
gfCNCPoint3[25884] = {X 371.5193, Y 53.9200, Z -4.6667, A 0.000, B 0.000, C 0.000 }
gfCNCPoint3[25885] = {X 388.0597, Y 53.9200, Z -4.6667, A 0.000, B 0.000, C 0.000 }
gfCNCPoint3[25886] = {X 388.9676, Y 54.0223, Z -4.6667, A 0.000, B 0.000, C 0.000 }
gfCNCPoint3[25887] = {X 389.8299, Y 54.3240, Z -4.6667, A 0.000, B 0.000, C 0.000 }
gfCNCPoint3[25888] = {X 390.6035, Y 54.8101, Z -4.6667, A 0.000, B 0.000, C 0.000 }
gfCNCPoint3[25889] = {X 391.2496, Y 55.4562, Z -4.6667, A 0.000, B 0.000, C 0.000 }
gfCNCPoint3[25890] = {X 391.7356, Y 56.2298, Z -4.6667, A 0.000, B 0.000, C 0.000 }
gfCNCPoint3[25891] = {X 392.0374, Y 57.0921, Z -4.6667, A 0.000, B 0.000, C 0.000 }
gfCNCPoint3[25892] = {X 392.1397, Y 58.0000, Z -4.6667, A 0.000, B 0.000, C 0.000 }
gfCNCPoint3[25893] = {X 392.1397, Y 58.9342, Z -4.6667, A 0.000, B 0.000, C 0.000 }
gfCNCPoint3[25894] = {X 392.0323, Y 59.8641, Z -4.6667, A 0.000, B 0.000, C 0.000 }
gfCNCPoint3[25895] = {X 391.7158, Y 60.7450, Z -4.6667, A 0.000, B 0.000, C 0.000 }
gfCNCPoint3[25896] = {X 391.1828, Y 61.5604, Z -4.6667, A 0.000, B 0.000, C 0.000 }
gfCNCPoint3[25897] = {X 390.4726, Y 62.2272, Z -4.6667, A 0.000, B 0.000, C 0.000 }
gfCNCPoint3[25898] = {X 389.6252, Y 62.7077, Z -4.6667, A 0.000, B 0.000, C 0.000 }
gfCNCPoint3[25899] = {X 388.6884, Y 62.9748, Z -4.6667, A 0.000, B 0.000, C 0.000 }
gfCNCPoint3[25900] = {X 388.5551, Y 62.9939, Z -4.6667, A 0.000, B 0.000, C 0.000 }
gfCNCPoint3[25901] = {X 388.4213, Y 63.0087, Z -4.6667, A 0.000, B 0.000, C 0.000 }
gfCNCPoint3[25902] = {X 388.4190, Y 63.1547, Z -4.6667, A 0.000, B 0.000, C 0.000 }
gfCNCPoint3[25903] = {X 388.4169, Y 84.6157, Z -4.6667, A 0.000, B 0.000, C 0.000 }
gfCNCPoint3[25904] = {X 388.3578, Y 86.2534, Z -4.6667, A 0.000, B 0.000, C 0.000 }
gfCNCPoint3[25905] = {X 388.1561, Y 87.8797, Z -4.6667, A 0.000, B 0.000, C 0.000 }
gfCNCPoint3[25906] = {X 387.8132, Y 89.4822, Z -4.6667, A 0.000, B 0.000, C 0.000 }
gfCNCPoint3[25907] = {X 387.2918, Y 91.0375, Z -4.6667, A 0.000, B 0.000, C 0.000 }
gfCNCPoint3[25908] = {X 386.5573, Y 92.5044, Z -4.6667, A 0.000, B 0.000, C 0.000 }
gfCNCPoint3[25909] = {X 385.6244, Y 93.8538, Z -4.6667, A 0.000, B 0.000, C 0.000 }
gfCNCPoint3[25910] = {X 384.5114, Y 95.0589, Z -4.6667, A 0.000, B 0.000, C 0.000 }
gfCNCPoint3[25911] = {X 383.0165, Y 96.3185, Z -4.6667, A 0.000, B 0.000, C 0.000 }
gfCNCPoint3[25912] = {X 381.3964, Y 97.4123, Z -4.6667, A 0.000, B 0.000, C 0.000 }
gfCNCPoint3[25913] = {X 379.6693, Y 98.3279, Z -4.6667, A 0.000, B 0.000, C 0.000 }
gfCNCPoint3[25914] = {X 377.4141, Y 99.2773, Z -4.6667, A 0.000, B 0.000, C 0.000 }
gfCNCPoint3[25915] = {X 375.0963, Y 100.0620, Z -4.6667, A 0.000, B 0.000, C 0.000 }
gfCNCPoint3[25916] = {X 372.7282, Y 100.6780, Z -4.6667, A 0.000, B 0.000, C 0.000 }
gfCNCPoint3[25917] = {X 368.8293, Y 101.4298, Z -4.6667, A 0.000, B 0.000, C 0.000 }
gfCNCPoint3[25918] = {X 364.8981, Y 101.9883, Z -4.6667, A 0.000, B 0.000, C 0.000 }
gfCNCPoint3[25919] = {X 360.9441, Y 102.3524, Z -4.6667, A 0.000, B 0.000, C 0.000 }
gfCNCPoint3[25920] = {X 357.0920, Y 102.5770, Z -4.6667, A 0.000, B 0.000, C 0.000 }
gfCNCPoint3[25921] = {X 353.2361, Y 102.7222, Z -4.6667, A 0.000, B 0.000, C 0.000 }
gfCNCPoint3[25922] = {X 353.3454, Y 106.7207, Z -4.6667, A 0.000, B 0.000, C 0.000 }
gfCNCPoint3[25923] = {X 353.2339, Y 102.6422, Z -4.6667, A 0.000, B 0.000, C 0.000 }
gfCNCPoint3[25924] = {X 348.1836, Y 102.7119, Z -4.6667, A 0.000, B 0.000, C 0.000 }
gfCNCPoint3[25925] = {X 343.1333, Y 102.6453, Z -4.6667, A 0.000, B 0.000, C 0.000 }
gfCNCPoint3[25926] = {X 338.0866, Y 102.4422, Z -4.6667, A 0.000, B 0.000, C 0.000 }
gfCNCPoint3[25927] = {X 334.1453, Y 102.1662, Z -4.6667, A 0.000, B 0.000, C 0.000 }
gfCNCPoint3[25928] = {X 330.2189, Y 101.7258, Z -4.6667, A 0.000, B 0.000, C 0.000 }
gfCNCPoint3[25929] = {X 326.3144, Y 101.1218, Z -4.6667, A 0.000, B 0.000, C 0.000 }
gfCNCPoint3[25930] = {X 323.4874, Y 100.5228, Z -4.6667, A 0.000, B 0.000, C 0.000 }
gfCNCPoint3[25931] = {X 320.7124, Y 99.7164, Z -4.6667, A 0.000, B 0.000, C 0.000 }
gfCNCPoint3[25932] = {X 318.0046, Y 98.7069, Z -4.6667, A 0.000, B 0.000, C 0.000 }
gfCNCPoint3[25933] = {X 316.5163, Y 98.0195, Z -4.6667, A 0.000, B 0.000, C 0.000 }
gfCNCPoint3[25934] = {X 315.0903, Y 97.2105, Z -4.6667, A 0.000, B 0.000, C 0.000 }
gfCNCPoint3[25935] = {X 313.7367, Y 96.2857, Z -4.6667, A 0.000, B 0.000, C 0.000 }
gfCNCPoint3[25936] = {X 312.4647, Y 95.2514, Z -4.6667, A 0.000, B 0.000, C 0.000 }
gfCNCPoint3[25937] = {X 311.4878, Y 94.2797, Z -4.6667, A 0.000, B 0.000, C 0.000 }
gfCNCPoint3[25938] = {X 310.6331, Y 93.1991, Z -4.6667, A 0.000, B 0.000, C 0.000 }
gfCNCPoint3[25939] = {X 309.9125, Y 92.0247, Z -4.6667, A 0.000, B 0.000, C 0.000 }
gfCNCPoint3[25940] = {X 309.3362, Y 90.7732, Z -4.6667, A 0.000, B 0.000, C 0.000 }
gfCNCPoint3[25941] = {X 308.9124, Y 89.4621, Z -4.6667, A 0.000, B 0.000, C 0.000 }
gfCNCPoint3[25942] = {X 308.5747, Y 87.8658, Z -4.6667, A 0.000, B 0.000, C 0.000 }
gfCNCPoint3[25943] = {X 308.3752, Y 86.2464, Z -4.6667, A 0.000, B 0.000, C 0.000 }
gfCNCPoint3[25944] = {X 308.3154, Y 84.6159, Z -4.6667, A 0.000, B 0.000, C 0.000 }
gfCNCPoint3[25945] = {X 308.3166, Y 62.9243, Z -4.6667, A 0.000, B 0.000, C 0.000 }
gfCNCPoint3[25946] = {X 307.4741, Y 62.7734, Z -4.6667, A 0.000, B 0.000, C 0.000 }
gfCNCPoint3[25947] = {X 306.6829, Y 62.4468, Z -4.6667, A 0.000, B 0.000, C 0.000 }
gfCNCPoint3[25948] = {X 305.9793, Y 61.9592, Z -4.6667, A 0.000, B 0.000, C 0.000 }
gfCNCPoint3[25949] = {X 305.3955, Y 61.3332, Z -4.6667, A 0.000, B 0.000, C 0.000 }
gfCNCPoint3[25950] = {X 304.9584, Y 60.5972, Z -4.6667, A 0.000, B 0.000, C 0.000 }
gfCNCPoint3[25951] = {X 304.6878, Y 59.7851, Z -4.6667, A 0.000, B 0.000, C 0.000 }
gfCNCPoint3[25952] = {X 304.5962, Y 58.9341, Z -4.6667, A 0.000, B 0.000, C 0.000 }
gfCNCPoint3[25953] = {X 304.5962, Y 58.0000, Z -4.6667, A 0.000, B 0.000, C 0.000 }
gfCNCPoint3[25954] = {X 304.6965, Y 57.1099, Z -4.6667, A 0.000, B 0.000, C 0.000 }
gfCNCPoint3[25955] = {X 304.9923, Y 56.2645, Z -4.6667, A 0.000, B 0.000, C 0.000 }
gfCNCPoint3[25956] = {X 305.4689, Y 55.5060, Z -4.6667, A 0.000, B 0.000, C 0.000 }
gfCNCPoint3[25957] = {X 306.1023, Y 54.8727, Z -4.6667, A 0.000, B 0.000, C 0.000 }
gfCNCPoint3[25958] = {X 306.8607, Y 54.3961, Z -4.6667, A 0.000, B 0.000, C 0.000 }
gfCNCPoint3[25959] = {X 307.7061, Y 54.1003, Z -4.6667, A 0.000, B 0.000, C 0.000 }
gfCNCPoint3[25960] = {X 308.5962, Y 54.0000, Z -4.6667, A 0.000, B 0.000, C 0.000 }
gfCNCPoint3[25961] = {X 324.3107, Y 54.0000, Z -4.6667, A 0.000, B 0.000, C 0.000 }
gfCNCPoint3[25962] = {X 325.2008, Y 54.1003, Z -4.6667, A 0.000, B 0.000, C 0.000 }
gfCNCPoint3[25963] = {X 326.0462, Y 54.3961, Z -4.6667, A 0.000, B 0.000, C 0.000 }
gfCNCPoint3[25964] = {X 326.8046, Y 54.8727, Z -4.6667, A 0.000, B 0.000, C 0.000 }
gfCNCPoint3[25965] = {X 327.4380, Y 55.5060, Z -4.6667, A 0.000, B 0.000, C 0.000 }
gfCNCPoint3[25966] = {X 327.9146, Y 56.2645, Z -4.6667, A 0.000, B 0.000, C 0.000 }
gfCNCPoint3[25967] = {X 328.2104, Y 57.1099, Z -4.6667, A 0.000, B 0.000, C 0.000 }
gfCNCPoint3[25968] = {X 328.3107, Y 58.0000, Z -4.6667, A 0.000, B 0.000, C 0.000 }
gfCNCPoint3[25969] = {X 328.3107, Y 58.9341, Z -4.6667, A 0.000, B 0.000, C 0.000 }
gfCNCPoint3[25970] = {X 328.2152, Y 59.7844, Z -4.6667, A 0.000, B 0.000, C 0.000 }
gfCNCPoint3[25971] = {X 327.9427, Y 60.5955, Z -4.6667, A 0.000, B 0.000, C 0.000 }
gfCNCPoint3[25972] = {X 327.5054, Y 61.3310, Z -4.6667, A 0.000, B 0.000, C 0.000 }
gfCNCPoint3[25973] = {X 326.9229, Y 61.9579, Z -4.6667, A 0.000, B 0.000, C 0.000 }
gfCNCPoint3[25974] = {X 326.2215, Y 62.4479, Z -4.6667, A 0.000, B 0.000, C 0.000 }
gfCNCPoint3[25975] = {X 325.4326, Y 62.7792, Z -4.6667, A 0.000, B 0.000, C 0.000 }
gfCNCPoint3[25976] = {X 324.5915, Y 62.9368, Z -4.6667, A 0.000, B 0.000, C 0.000 }
gfCNCPoint3[25977] = {X 324.5932, Y 83.2313, Z -4.6667, A 0.000, B 0.000, C 0.000 }
gfCNCPoint3[25978] = {X 324.6068, Y 84.6159, Z -4.6667, A 0.000, B 0.000, C 0.000 }
gfCNCPoint3[25979] = {X 324.6902, Y 85.9180, Z -4.6667, A 0.000, B 0.000, C 0.000 }
gfCNCPoint3[25980] = {X 324.9294, Y 87.2007, Z -4.6667, A 0.000, B 0.000, C 0.000 }
gfCNCPoint3[25981] = {X 325.2359, Y 87.5550, Z -4.6667, A 0.000, B 0.000, C 0.000 }
gfCNCPoint3[25982] = {X 325.6219, Y 87.8206, Z -4.6667, A 0.000, B 0.000, C 0.000 }
gfCNCPoint3[25983] = {X 326.0763, Y 88.0775, Z -4.6667, A 0.000, B 0.000, C 0.000 }
gfCNCPoint3[25984] = {X 327.5511, Y 88.6904, Z -4.6667, A 0.000, B 0.000, C 0.000 }
gfCNCPoint3[25985] = {X 329.0843, Y 89.1377, Z -4.6667, A 0.000, B 0.000, C 0.000 }
gfCNCPoint3[25986] = {X 332.1822, Y 89.7578, Z -4.6667, A 0.000, B 0.000, C 0.000 }
gfCNCPoint3[25987] = {X 335.3167, Y 90.1536, Z -4.6667, A 0.000, B 0.000, C 0.000 }
gfCNCPoint3[25988] = {X 339.4647, Y 90.4743, Z -4.6667, A 0.000, B 0.000, C 0.000 }
gfCNCPoint3[25989] = {X 343.6212, Y 90.6543, Z -4.6667, A 0.000, B 0.000, C 0.000 }
gfCNCPoint3[25990] = {X 347.7814, Y 90.6934, Z -4.6667, A 0.000, B 0.000, C 0.000 }
gfCNCPoint3[25991] = {X 352.1732, Y 90.6548, Z -4.6667, A 0.000, B 0.000, C 0.000 }
gfCNCPoint3[25992] = {X 356.5609, Y 90.4584, Z -4.6667, A 0.000, B 0.000, C 0.000 }
gfCNCPoint3[25993] = {X 360.9386, Y 90.1045, Z -4.6667, A 0.000, B 0.000, C 0.000 }
gfCNCPoint3[25994] = {X 363.2713, Y 89.8143, Z -4.6667, A 0.000, B 0.000, C 0.000 }
gfCNCPoint3[25995] = {X 365.5824, Y 89.3845, Z -4.6667, A 0.000, B 0.000, C 0.000 }
gfCNCPoint3[25996] = {X 367.8634, Y 88.8165, Z -4.6667, A 0.000, B 0.000, C 0.000 }
gfCNCPoint3[25997] = {X 368.8287, Y 88.4919, Z -4.6667, A 0.000, B 0.000, C 0.000 }
gfCNCPoint3[25998] = {X 369.7516, Y 88.0610, Z -4.6667, A 0.000, B 0.000, C 0.000 }
gfCNCPoint3[25999] = {X 370.6203, Y 87.5295, Z -4.6667, A 0.000, B 0.000, C 0.000 }
gfCNCPoint3[26000] = {X 370.8582, Y 87.2819, Z -4.6667, A 0.000, B 0.000, C 0.000 }
gfCNCPoint3[26001] = {X 370.9809, Y 86.9612, Z -4.6667, A 0.000, B 0.000, C 0.000 }
gfCNCPoint3[26002] = {X 371.1752, Y 85.4001, Z -4.6667, A 0.000, B 0.000, C 0.000 }
gfCNCPoint3[26003] = {X 371.2401, Y 83.8283, Z -4.6667, A 0.000, B 0.000, C 0.000 }
gfCNCPoint3[26004] = {X 371.2386, Y 63.0392, Z -4.6667, A 0.000, B 0.000, C 0.000 }
gfCNCPoint3[26005] = {X 371.2440, Y 62.9246, Z -4.6667, A 0.000, B 0.000, C 0.000 }
gfCNCPoint3[26006] = {X 371.0719, Y 62.9090, Z -4.6667, A 0.000, B 0.000, C 0.000 }
gfCNCPoint3[26007] = {X 370.9005, Y 62.8859, Z -4.6667, A 0.000, B 0.000, C 0.000 }
gfCNCPoint3[26008] = {X 369.9940, Y 62.6318, Z -4.6667, A 0.000, B 0.000, C 0.000 }
gfCNCPoint3[26009] = {X 369.1719, Y 62.1729, Z -4.6667, A 0.000, B 0.000, C 0.000 }
gfCNCPoint3[26010] = {X 368.4799, Y 61.5345, Z -4.6667, A 0.000, B 0.000, C 0.000 }
gfCNCPoint3[26011] = {X 367.9563, Y 60.7521, Z -4.6667, A 0.000, B 0.000, C 0.000 }
gfCNCPoint3[26012] = {X 367.6301, Y 59.8690, Z -4.6667, A 0.000, B 0.000, C 0.000 }
gfCNCPoint3[26013] = {X 367.5193, Y 58.9340, Z -4.6667, A 0.000, B 0.000, C 0.000 }
gfCNCPoint3[26014] = {X 367.5193, Y 58.0000, Z -4.6667, A 0.000, B 0.000, C 0.000 }
gfCNCPoint3[26015] = {X 367.6196, Y 57.1099, Z -4.6667, A 0.000, B 0.000, C 0.000 }
gfCNCPoint3[26016] = {X 367.9154, Y 56.2645, Z -4.6667, A 0.000, B 0.000, C 0.000 }
gfCNCPoint3[26017] = {X 368.3920, Y 55.5060, Z -4.6667, A 0.000, B 0.000, C 0.000 }
gfCNCPoint3[26018] = {X 369.0253, Y 54.8727, Z -4.6667, A 0.000, B 0.000, C 0.000 }
gfCNCPoint3[26019] = {X 369.7837, Y 54.3961, Z -4.6667, A 0.000, B 0.000, C 0.000 }
gfCNCPoint3[26020] = {X 370.6292, Y 54.1003, Z -4.6667, A 0.000, B 0.000, C 0.000 }
gfCNCPoint3[26021] = {X 371.5193, Y 54.0000, Z -4.6667, A 0.000, B 0.000, C 0.000 }
gfCNCPoint3[26022] = {X 388.0597, Y 54.0000, Z -4.6667, A 0.000, B 0.000, C 0.000 }
gfCNCPoint3[26023] = {X 388.9498, Y 54.1003, Z -4.6667, A 0.000, B 0.000, C 0.000 }
gfCNCPoint3[26024] = {X 389.7952, Y 54.3961, Z -4.6667, A 0.000, B 0.000, C 0.000 }
gfCNCPoint3[26025] = {X 390.5536, Y 54.8727, Z -4.6667, A 0.000, B 0.000, C 0.000 }
gfCNCPoint3[26026] = {X 391.1870, Y 55.5060, Z -4.6667, A 0.000, B 0.000, C 0.000 }
gfCNCPoint3[26027] = {X 391.6636, Y 56.2645, Z -4.6667, A 0.000, B 0.000, C 0.000 }
gfCNCPoint3[26028] = {X 391.9594, Y 57.1099, Z -4.6667, A 0.000, B 0.000, C 0.000 }
gfCNCPoint3[26029] = {X 392.0597, Y 58.0000, Z -4.6667, A 0.000, B 0.000, C 0.000 }
gfCNCPoint3[26030] = {X 392.0595, Y 58.9671, Z -4.6667, A 0.000, B 0.000, C 0.000 }
gfCNCPoint3[26031] = {X 391.9506, Y 59.8618, Z -4.6667, A 0.000, B 0.000, C 0.000 }
gfCNCPoint3[26032] = {X 391.6441, Y 60.7094, Z -4.6667, A 0.000, B 0.000, C 0.000 }
gfCNCPoint3[26033] = {X 391.1215, Y 61.5090, Z -4.6667, A 0.000, B 0.000, C 0.000 }
gfCNCPoint3[26034] = {X 390.4252, Y 62.1628, Z -4.6667, A 0.000, B 0.000, C 0.000 }
gfCNCPoint3[26035] = {X 389.5943, Y 62.6339, Z -4.6667, A 0.000, B 0.000, C 0.000 }
gfCNCPoint3[26036] = {X 388.6757, Y 62.8958, Z -4.6667, A 0.000, B 0.000, C 0.000 }
gfCNCPoint3[26037] = {X 388.5095, Y 62.9189, Z -4.6667, A 0.000, B 0.000, C 0.000 }
gfCNCPoint3[26038] = {X 388.3425, Y 62.9350, Z -4.6667, A 0.000, B 0.000, C 0.000 }
gfCNCPoint3[26039] = {X 388.3390, Y 63.1540, Z -4.6667, A 0.000, B 0.000, C 0.000 }
gfCNCPoint3[26040] = {X 388.3390, Y 83.9236, Z -4.6667, A 0.000, B 0.000, C 0.000 }
gfCNCPoint3[26041] = {X 388.3369, Y 84.6159, Z -4.6667, A 0.000, B 0.000, C 0.000 }
gfCNCPoint3[26042] = {X 388.2781, Y 86.2468, Z -4.6667, A 0.000, B 0.000, C 0.000 }
gfCNCPoint3[26043] = {X 388.0772, Y 87.8663, Z -4.6667, A 0.000, B 0.000, C 0.000 }
gfCNCPoint3[26044] = {X 387.7357, Y 89.4621, Z -4.6667, A 0.000, B 0.000, C 0.000 }
gfCNCPoint3[26045] = {X 387.2179, Y 91.0068, Z -4.6667, A 0.000, B 0.000, C 0.000 }
gfCNCPoint3[26046] = {X 386.4885, Y 92.4637, Z -4.6667, A 0.000, B 0.000, C 0.000 }
gfCNCPoint3[26047] = {X 385.5619, Y 93.8038, Z -4.6667, A 0.000, B 0.000, C 0.000 }
gfCNCPoint3[26048] = {X 384.4566, Y 95.0007, Z -4.6667, A 0.000, B 0.000, C 0.000 }
gfCNCPoint3[26049] = {X 382.9683, Y 96.2547, Z -4.6667, A 0.000, B 0.000, C 0.000 }
gfCNCPoint3[26050] = {X 381.3552, Y 97.3437, Z -4.6667, A 0.000, B 0.000, C 0.000 }
gfCNCPoint3[26051] = {X 379.6357, Y 98.2553, Z -4.6667, A 0.000, B 0.000, C 0.000 }
gfCNCPoint3[26052] = {X 377.3857, Y 99.2025, Z -4.6667, A 0.000, B 0.000, C 0.000 }
gfCNCPoint3[26053] = {X 375.0734, Y 99.9854, Z -4.6667, A 0.000, B 0.000, C 0.000 }
gfCNCPoint3[26054] = {X 372.7108, Y 100.5999, Z -4.6667, A 0.000, B 0.000, C 0.000 }
gfCNCPoint3[26055] = {X 368.8159, Y 101.3509, Z -4.6667, A 0.000, B 0.000, C 0.000 }
gfCNCPoint3[26056] = {X 364.8886, Y 101.9089, Z -4.6667, A 0.000, B 0.000, C 0.000 }
gfCNCPoint3[26057] = {X 360.9386, Y 102.2725, Z -4.6667, A 0.000, B 0.000, C 0.000 }
gfCNCPoint3[26058] = {X 357.0882, Y 102.4971, Z -4.6667, A 0.000, B 0.000, C 0.000 }
gfCNCPoint3[26059] = {X 353.2339, Y 102.6422, Z -4.6667, A 0.000, B 0.000, C 0.000 }
gfCNCPoint3[26060] = {X 353.3454, Y 106.7207, Z -4.6667, A 0.000, B 0.000, C 0.000 }
gfCNCPoint3[26061] = {X 353.3454, Y 106.7207, Z -1.6667, A 0.000, B 0.000, C 0.000 }
gfCNCPoint3[26062] = {X 353.3454, Y 106.7207, Z 11.0000, A 0.000, B 0.000, C 0.000 }
gfCNCPoint3[26063] = {X 411.5988, Y 79.5927, Z 11.0000, A 0.000, B 0.000, C 0.000 }
gfCNCPoint3[26064] = {X 411.5988, Y 79.5927, Z -1.6667, A 0.000, B 0.000, C 0.000 }
gfCNCPoint3[26065] = {X 411.5988, Y 79.5927, Z -4.6667, A 0.000, B 0.000, C 0.000 }
gfCNCPoint3[26066] = {X 413.7991, Y 83.0285, Z -4.6667, A 0.000, B 0.000, C 0.000 }
gfCNCPoint3[26067] = {X 428.0545, Y 73.8995, Z -4.6667, A 0.000, B 0.000, C 0.000 }
gfCNCPoint3[26068] = {X 403.7555, Y 64.3658, Z -4.6667, A 0.000, B 0.000, C 0.000 }
gfCNCPoint3[26069] = {X 402.0596, Y 63.8044, Z -4.6667, A 0.000, B 0.000, C 0.000 }
gfCNCPoint3[26070] = {X 400.3123, Y 63.4322, Z -4.6667, A 0.000, B 0.000, C 0.000 }
gfCNCPoint3[26071] = {X 398.5348, Y 63.2540, Z -4.6667, A 0.000, B 0.000, C 0.000 }
gfCNCPoint3[26072] = {X 397.5823, Y 63.1425, Z -4.6667, A 0.000, B 0.000, C 0.000 }
gfCNCPoint3[26073] = {X 396.6778, Y 62.8236, Z -4.6667, A 0.000, B 0.000, C 0.000 }
gfCNCPoint3[26074] = {X 395.8660, Y 62.3129, Z -4.6667, A 0.000, B 0.000, C 0.000 }
gfCNCPoint3[26075] = {X 395.1868, Y 61.6358, Z -4.6667, A 0.000, B 0.000, C 0.000 }
gfCNCPoint3[26076] = {X 394.6738, Y 60.8255, Z -4.6667, A 0.000, B 0.000, C 0.000 }
gfCNCPoint3[26077] = {X 394.3522, Y 59.9220, Z -4.6667, A 0.000, B 0.000, C 0.000 }
gfCNCPoint3[26078] = {X 394.2379, Y 58.9697, Z -4.6667, A 0.000, B 0.000, C 0.000 }
gfCNCPoint3[26079] = {X 394.2377, Y 58.0000, Z -4.6667, A 0.000, B 0.000, C 0.000 }
gfCNCPoint3[26080] = {X 394.3460, Y 57.0387, Z -4.6667, A 0.000, B 0.000, C 0.000 }
gfCNCPoint3[26081] = {X 394.6655, Y 56.1256, Z -4.6667, A 0.000, B 0.000, C 0.000 }
gfCNCPoint3[26082] = {X 395.1802, Y 55.3065, Z -4.6667, A 0.000, B 0.000, C 0.000 }
gfCNCPoint3[26083] = {X 395.8642, Y 54.6225, Z -4.6667, A 0.000, B 0.000, C 0.000 }
gfCNCPoint3[26084] = {X 396.6833, Y 54.1078, Z -4.6667, A 0.000, B 0.000, C 0.000 }
gfCNCPoint3[26085] = {X 397.5964, Y 53.7883, Z -4.6667, A 0.000, B 0.000, C 0.000 }
gfCNCPoint3[26086] = {X 398.5577, Y 53.6800, Z -4.6667, A 0.000, B 0.000, C 0.000 }
gfCNCPoint3[26087] = {X 419.4886, Y 53.6800, Z -4.6667, A 0.000, B 0.000, C 0.000 }
gfCNCPoint3[26088] = {X 420.4499, Y 53.7883, Z -4.6667, A 0.000, B 0.000, C 0.000 }
gfCNCPoint3[26089] = {X 421.3630, Y 54.1078, Z -4.6667, A 0.000, B 0.000, C 0.000 }
gfCNCPoint3[26090] = {X 422.1821, Y 54.6225, Z -4.6667, A 0.000, B 0.000, C 0.000 }
gfCNCPoint3[26091] = {X 422.8661, Y 55.3065, Z -4.6667, A 0.000, B 0.000, C 0.000 }
gfCNCPoint3[26092] = {X 423.3808, Y 56.1256, Z -4.6667, A 0.000, B 0.000, C 0.000 }
gfCNCPoint3[26093] = {X 423.7003, Y 57.0387, Z -4.6667, A 0.000, B 0.000, C 0.000 }
gfCNCPoint3[26094] = {X 423.8086, Y 58.0000, Z -4.6667, A 0.000, B 0.000, C 0.000 }
gfCNCPoint3[26095] = {X 423.8086, Y 58.2321, Z -4.6667, A 0.000, B 0.000, C 0.000 }
gfCNCPoint3[26096] = {X 429.6116, Y 60.4934, Z -4.6667, A 0.000, B 0.000, C 0.000 }
gfCNCPoint3[26097] = {X 457.8586, Y 71.7006, Z -4.6667, A 0.000, B 0.000, C 0.000 }
gfCNCPoint3[26098] = {X 457.8607, Y 63.2123, Z -4.6667, A 0.000, B 0.000, C 0.000 }
gfCNCPoint3[26099] = {X 457.0090, Y 63.0032, Z -4.6667, A 0.000, B 0.000, C 0.000 }
gfCNCPoint3[26100] = {X 456.2171, Y 62.6265, Z -4.6667, A 0.000, B 0.000, C 0.000 }
gfCNCPoint3[26101] = {X 455.5177, Y 62.0975, Z -4.6667, A 0.000, B 0.000, C 0.000 }
gfCNCPoint3[26102] = {X 454.9394, Y 61.4382, Z -4.6667, A 0.000, B 0.000, C 0.000 }
gfCNCPoint3[26103] = {X 454.5062, Y 60.6757, Z -4.6667, A 0.000, B 0.000, C 0.000 }
gfCNCPoint3[26104] = {X 454.2360, Y 59.8414, Z -4.6667, A 0.000, B 0.000, C 0.000 }
gfCNCPoint3[26105] = {X 454.1398, Y 58.9697, Z -4.6667, A 0.000, B 0.000, C 0.000 }
gfCNCPoint3[26106] = {X 454.1396, Y 58.0000, Z -4.6667, A 0.000, B 0.000, C 0.000 }
gfCNCPoint3[26107] = {X 454.2479, Y 57.0387, Z -4.6667, A 0.000, B 0.000, C 0.000 }
gfCNCPoint3[26108] = {X 454.5674, Y 56.1256, Z -4.6667, A 0.000, B 0.000, C 0.000 }
gfCNCPoint3[26109] = {X 455.0821, Y 55.3065, Z -4.6667, A 0.000, B 0.000, C 0.000 }
gfCNCPoint3[26110] = {X 455.7661, Y 54.6225, Z -4.6667, A 0.000, B 0.000, C 0.000 }
gfCNCPoint3[26111] = {X 456.5852, Y 54.1078, Z -4.6667, A 0.000, B 0.000, C 0.000 }
gfCNCPoint3[26112] = {X 457.4983, Y 53.7883, Z -4.6667, A 0.000, B 0.000, C 0.000 }
gfCNCPoint3[26113] = {X 458.4596, Y 53.6800, Z -4.6667, A 0.000, B 0.000, C 0.000 }
gfCNCPoint3[26114] = {X 475.0000, Y 53.6800, Z -4.6667, A 0.000, B 0.000, C 0.000 }
gfCNCPoint3[26115] = {X 475.9613, Y 53.7883, Z -4.6667, A 0.000, B 0.000, C 0.000 }
gfCNCPoint3[26116] = {X 476.8744, Y 54.1078, Z -4.6667, A 0.000, B 0.000, C 0.000 }
gfCNCPoint3[26117] = {X 477.6935, Y 54.6225, Z -4.6667, A 0.000, B 0.000, C 0.000 }
gfCNCPoint3[26118] = {X 478.3775, Y 55.3065, Z -4.6667, A 0.000, B 0.000, C 0.000 }
gfCNCPoint3[26119] = {X 478.8922, Y 56.1256, Z -4.6667, A 0.000, B 0.000, C 0.000 }
gfCNCPoint3[26120] = {X 479.2117, Y 57.0387, Z -4.6667, A 0.000, B 0.000, C 0.000 }
gfCNCPoint3[26121] = {X 479.3200, Y 58.0000, Z -4.6667, A 0.000, B 0.000, C 0.000 }
gfCNCPoint3[26122] = {X 479.3200, Y 58.9342, Z -4.6667, A 0.000, B 0.000, C 0.000 }
gfCNCPoint3[26123] = {X 479.2300, Y 59.8114, Z -4.6667, A 0.000, B 0.000, C 0.000 }
gfCNCPoint3[26124] = {X 478.9637, Y 60.6521, Z -4.6667, A 0.000, B 0.000, C 0.000 }
gfCNCPoint3[26125] = {X 478.5322, Y 61.4212, Z -4.6667, A 0.000, B 0.000, C 0.000 }
gfCNCPoint3[26126] = {X 477.9536, Y 62.0866, Z -4.6667, A 0.000, B 0.000, C 0.000 }
gfCNCPoint3[26127] = {X 477.2519, Y 62.6207, Z -4.6667, A 0.000, B 0.000, C 0.000 }
gfCNCPoint3[26128] = {X 476.4564, Y 63.0012, Z -4.6667, A 0.000, B 0.000, C 0.000 }
gfCNCPoint3[26129] = {X 475.6002, Y 63.2122, Z -4.6667, A 0.000, B 0.000, C 0.000 }
gfCNCPoint3[26130] = {X 475.6007, Y 92.7681, Z -4.6667, A 0.000, B 0.000, C 0.000 }
gfCNCPoint3[26131] = {X 475.9972, Y 92.8673, Z -4.6667, A 0.000, B 0.000, C 0.000 }
gfCNCPoint3[26132] = {X 476.3881, Y 92.9868, Z -4.6667, A 0.000, B 0.000, C 0.000 }
gfCNCPoint3[26133] = {X 477.1997, Y 93.3557, Z -4.6667, A 0.000, B 0.000, C 0.000 }
gfCNCPoint3[26134] = {X 477.9175, Y 93.8842, Z -4.6667, A 0.000, B 0.000, C 0.000 }
gfCNCPoint3[26135] = {X 478.5108, Y 94.5496, Z -4.6667, A 0.000, B 0.000, C 0.000 }
gfCNCPoint3[26136] = {X 478.9538, Y 95.3232, Z -4.6667, A 0.000, B 0.000, C 0.000 }
gfCNCPoint3[26137] = {X 479.2274, Y 96.1716, Z -4.6667, A 0.000, B 0.000, C 0.000 }
gfCNCPoint3[26138] = {X 479.3200, Y 97.0582, Z -4.6667, A 0.000, B 0.000, C 0.000 }
gfCNCPoint3[26139] = {X 479.3200, Y 98.0000, Z -4.6667, A 0.000, B 0.000, C 0.000 }
gfCNCPoint3[26140] = {X 479.2117, Y 98.9613, Z -4.6667, A 0.000, B 0.000, C 0.000 }
gfCNCPoint3[26141] = {X 478.8922, Y 99.8744, Z -4.6667, A 0.000, B 0.000, C 0.000 }
gfCNCPoint3[26142] = {X 478.3775, Y 100.6935, Z -4.6667, A 0.000, B 0.000, C 0.000 }
gfCNCPoint3[26143] = {X 477.6935, Y 101.3775, Z -4.6667, A 0.000, B 0.000, C 0.000 }
gfCNCPoint3[26144] = {X 476.8744, Y 101.8922, Z -4.6667, A 0.000, B 0.000, C 0.000 }
gfCNCPoint3[26145] = {X 475.9613, Y 102.2117, Z -4.6667, A 0.000, B 0.000, C 0.000 }
gfCNCPoint3[26146] = {X 475.0000, Y 102.3200, Z -4.6667, A 0.000, B 0.000, C 0.000 }
gfCNCPoint3[26147] = {X 458.4596, Y 102.3200, Z -4.6667, A 0.000, B 0.000, C 0.000 }
gfCNCPoint3[26148] = {X 457.4983, Y 102.2117, Z -4.6667, A 0.000, B 0.000, C 0.000 }
gfCNCPoint3[26149] = {X 456.5852, Y 101.8922, Z -4.6667, A 0.000, B 0.000, C 0.000 }
gfCNCPoint3[26150] = {X 455.7661, Y 101.3775, Z -4.6667, A 0.000, B 0.000, C 0.000 }
gfCNCPoint3[26151] = {X 455.0821, Y 100.6935, Z -4.6667, A 0.000, B 0.000, C 0.000 }
gfCNCPoint3[26152] = {X 454.5674, Y 99.8744, Z -4.6667, A 0.000, B 0.000, C 0.000 }
gfCNCPoint3[26153] = {X 454.2479, Y 98.9613, Z -4.6667, A 0.000, B 0.000, C 0.000 }
gfCNCPoint3[26154] = {X 454.1396, Y 98.0000, Z -4.6667, A 0.000, B 0.000, C 0.000 }
gfCNCPoint3[26155] = {X 454.1396, Y 97.0659, Z -4.6667, A 0.000, B 0.000, C 0.000 }
gfCNCPoint3[26156] = {X 454.2295, Y 96.1891, Z -4.6667, A 0.000, B 0.000, C 0.000 }
gfCNCPoint3[26157] = {X 454.4955, Y 95.3488, Z -4.6667, A 0.000, B 0.000, C 0.000 }
gfCNCPoint3[26158] = {X 454.9265, Y 94.5800, Z -4.6667, A 0.000, B 0.000, C 0.000 }
gfCNCPoint3[26159] = {X 455.5046, Y 93.9147, Z -4.6667, A 0.000, B 0.000, C 0.000 }
gfCNCPoint3[26160] = {X 456.2057, Y 93.3805, Z -4.6667, A 0.000, B 0.000, C 0.000 }
gfCNCPoint3[26161] = {X 457.0006, Y 92.9998, Z -4.6667, A 0.000, B 0.000, C 0.000 }
gfCNCPoint3[26162] = {X 457.8563, Y 92.7883, Z -4.6667, A 0.000, B 0.000, C 0.000 }
gfCNCPoint3[26163] = {X 457.8563, Y 85.5950, Z -4.6667, A 0.000, B 0.000, C 0.000 }
gfCNCPoint3[26164] = {X 444.8591, Y 80.5001, Z -4.6667, A 0.000, B 0.000, C 0.000 }
gfCNCPoint3[26165] = {X 420.0235, Y 96.5883, Z -4.6667, A 0.000, B 0.000, C 0.000 }
gfCNCPoint3[26166] = {X 420.0267, Y 97.0648, Z -4.6667, A 0.000, B 0.000, C 0.000 }
gfCNCPoint3[26167] = {X 420.0267, Y 98.0000, Z -4.6667, A 0.000, B 0.000, C 0.000 }
gfCNCPoint3[26168] = {X 419.9184, Y 98.9613, Z -4.6667, A 0.000, B 0.000, C 0.000 }
gfCNCPoint3[26169] = {X 419.5989, Y 99.8744, Z -4.6667, A 0.000, B 0.000, C 0.000 }
gfCNCPoint3[26170] = {X 419.0842, Y 100.6935, Z -4.6667, A 0.000, B 0.000, C 0.000 }
gfCNCPoint3[26171] = {X 418.4002, Y 101.3775, Z -4.6667, A 0.000, B 0.000, C 0.000 }
gfCNCPoint3[26172] = {X 417.5811, Y 101.8922, Z -4.6667, A 0.000, B 0.000, C 0.000 }
gfCNCPoint3[26173] = {X 416.6680, Y 102.2117, Z -4.6667, A 0.000, B 0.000, C 0.000 }
gfCNCPoint3[26174] = {X 415.7067, Y 102.3200, Z -4.6667, A 0.000, B 0.000, C 0.000 }
gfCNCPoint3[26175] = {X 396.4059, Y 102.3200, Z -4.6667, A 0.000, B 0.000, C 0.000 }
gfCNCPoint3[26176] = {X 395.4447, Y 102.2117, Z -4.6667, A 0.000, B 0.000, C 0.000 }
gfCNCPoint3[26177] = {X 394.5316, Y 101.8922, Z -4.6667, A 0.000, B 0.000, C 0.000 }
gfCNCPoint3[26178] = {X 393.7125, Y 101.3775, Z -4.6667, A 0.000, B 0.000, C 0.000 }
gfCNCPoint3[26179] = {X 393.0284, Y 100.6935, Z -4.6667, A 0.000, B 0.000, C 0.000 }
gfCNCPoint3[26180] = {X 392.5138, Y 99.8744, Z -4.6667, A 0.000, B 0.000, C 0.000 }
gfCNCPoint3[26181] = {X 392.1943, Y 98.9613, Z -4.6667, A 0.000, B 0.000, C 0.000 }
gfCNCPoint3[26182] = {X 392.0859, Y 98.0000, Z -4.6667, A 0.000, B 0.000, C 0.000 }
gfCNCPoint3[26183] = {X 392.0859, Y 97.0659, Z -4.6667, A 0.000, B 0.000, C 0.000 }
gfCNCPoint3[26184] = {X 392.1951, Y 96.1011, Z -4.6667, A 0.000, B 0.000, C 0.000 }
gfCNCPoint3[26185] = {X 392.5169, Y 95.1850, Z -4.6667, A 0.000, B 0.000, C 0.000 }
gfCNCPoint3[26186] = {X 393.0353, Y 94.3639, Z -4.6667, A 0.000, B 0.000, C 0.000 }
gfCNCPoint3[26187] = {X 393.7239, Y 93.6794, Z -4.6667, A 0.000, B 0.000, C 0.000 }
gfCNCPoint3[26188] = {X 394.5480, Y 93.1659, Z -4.6667, A 0.000, B 0.000, C 0.000 }
gfCNCPoint3[26189] = {X 395.4660, Y 92.8494, Z -4.6667, A 0.000, B 0.000, C 0.000 }
gfCNCPoint3[26190] = {X 396.4314, Y 92.7460, Z -4.6667, A 0.000, B 0.000, C 0.000 }
gfCNCPoint3[26191] = {X 397.3641, Y 92.7028, Z -4.6667, A 0.000, B 0.000, C 0.000 }
gfCNCPoint3[26192] = {X 398.2935, Y 92.6143, Z -4.6667, A 0.000, B 0.000, C 0.000 }
gfCNCPoint3[26193] = {X 398.9444, Y 92.4564, Z -4.6667, A 0.000, B 0.000, C 0.000 }
gfCNCPoint3[26194] = {X 399.5438, Y 92.1576, Z -4.6667, A 0.000, B 0.000, C 0.000 }
gfCNCPoint3[26195] = {X 413.7991, Y 83.0285, Z -4.6667, A 0.000, B 0.000, C 0.000 }
gfCNCPoint3[26196] = {X 411.6420, Y 79.6601, Z -4.6667, A 0.000, B 0.000, C 0.000 }
gfCNCPoint3[26197] = {X 413.8423, Y 83.0959, Z -4.6667, A 0.000, B 0.000, C 0.000 }
gfCNCPoint3[26198] = {X 428.2297, Y 73.8823, Z -4.6667, A 0.000, B 0.000, C 0.000 }
gfCNCPoint3[26199] = {X 403.7848, Y 64.2914, Z -4.6667, A 0.000, B 0.000, C 0.000 }
gfCNCPoint3[26200] = {X 402.0800, Y 63.7270, Z -4.6667, A 0.000, B 0.000, C 0.000 }
gfCNCPoint3[26201] = {X 400.3236, Y 63.3530, Z -4.6667, A 0.000, B 0.000, C 0.000 }
gfCNCPoint3[26202] = {X 398.5368, Y 63.1740, Z -4.6667, A 0.000, B 0.000, C 0.000 }
gfCNCPoint3[26203] = {X 397.6016, Y 63.0649, Z -4.6667, A 0.000, B 0.000, C 0.000 }
gfCNCPoint3[26204] = {X 396.7136, Y 62.7520, Z -4.6667, A 0.000, B 0.000, C 0.000 }
gfCNCPoint3[26205] = {X 395.9165, Y 62.2509, Z -4.6667, A 0.000, B 0.000, C 0.000 }
gfCNCPoint3[26206] = {X 395.2497, Y 61.5863, Z -4.6667, A 0.000, B 0.000, C 0.000 }
gfCNCPoint3[26207] = {X 394.7459, Y 60.7909, Z -4.6667, A 0.000, B 0.000, C 0.000 }
gfCNCPoint3[26208] = {X 394.4301, Y 59.9039, Z -4.6667, A 0.000, B 0.000, C 0.000 }
gfCNCPoint3[26209] = {X 394.3179, Y 58.9691, Z -4.6667, A 0.000, B 0.000, C 0.000 }
gfCNCPoint3[26210] = {X 394.3177, Y 58.0000, Z -4.6667, A 0.000, B 0.000, C 0.000 }
gfCNCPoint3[26211] = {X 394.4240, Y 57.0565, Z -4.6667, A 0.000, B 0.000, C 0.000 }
gfCNCPoint3[26212] = {X 394.7376, Y 56.1603, Z -4.6667, A 0.000, B 0.000, C 0.000 }
gfCNCPoint3[26213] = {X 395.2428, Y 55.3564, Z -4.6667, A 0.000, B 0.000, C 0.000 }
gfCNCPoint3[26214] = {X 395.9141, Y 54.6850, Z -4.6667, A 0.000, B 0.000, C 0.000 }
gfCNCPoint3[26215] = {X 396.7181, Y 54.1799, Z -4.6667, A 0.000, B 0.000, C 0.000 }
gfCNCPoint3[26216] = {X 397.6142, Y 53.8663, Z -4.6667, A 0.000, B 0.000, C 0.000 }
gfCNCPoint3[26217] = {X 398.5577, Y 53.7600, Z -4.6667, A 0.000, B 0.000, C 0.000 }
gfCNCPoint3[26218] = {X 419.4886, Y 53.7600, Z -4.6667, A 0.000, B 0.000, C 0.000 }
gfCNCPoint3[26219] = {X 420.4321, Y 53.8663, Z -4.6667, A 0.000, B 0.000, C 0.000 }
gfCNCPoint3[26220] = {X 421.3283, Y 54.1799, Z -4.6667, A 0.000, B 0.000, C 0.000 }
gfCNCPoint3[26221] = {X 422.1322, Y 54.6850, Z -4.6667, A 0.000, B 0.000, C 0.000 }
gfCNCPoint3[26222] = {X 422.8036, Y 55.3564, Z -4.6667, A 0.000, B 0.000, C 0.000 }
gfCNCPoint3[26223] = {X 423.3087, Y 56.1603, Z -4.6667, A 0.000, B 0.000, C 0.000 }
gfCNCPoint3[26224] = {X 423.6223, Y 57.0565, Z -4.6667, A 0.000, B 0.000, C 0.000 }
gfCNCPoint3[26225] = {X 423.7286, Y 58.0000, Z -4.6667, A 0.000, B 0.000, C 0.000 }
gfCNCPoint3[26226] = {X 423.7286, Y 58.2868, Z -4.6667, A 0.000, B 0.000, C 0.000 }
gfCNCPoint3[26227] = {X 429.5823, Y 60.5678, Z -4.6667, A 0.000, B 0.000, C 0.000 }
gfCNCPoint3[26228] = {X 457.9386, Y 71.8184, Z -4.6667, A 0.000, B 0.000, C 0.000 }
gfCNCPoint3[26229] = {X 457.9407, Y 63.1422, Z -4.6667, A 0.000, B 0.000, C 0.000 }
gfCNCPoint3[26230] = {X 457.0922, Y 62.9475, Z -4.6667, A 0.000, B 0.000, C 0.000 }
gfCNCPoint3[26231] = {X 456.3013, Y 62.5836, Z -4.6667, A 0.000, B 0.000, C 0.000 }
gfCNCPoint3[26232] = {X 455.6014, Y 62.0658, Z -4.6667, A 0.000, B 0.000, C 0.000 }
gfCNCPoint3[26233] = {X 455.0220, Y 61.4160, Z -4.6667, A 0.000, B 0.000, C 0.000 }
gfCNCPoint3[26234] = {X 454.5875, Y 60.6616, Z -4.6667, A 0.000, B 0.000, C 0.000 }
gfCNCPoint3[26235] = {X 454.3163, Y 59.8343, Z -4.6667, A 0.000, B 0.000, C 0.000 }
gfCNCPoint3[26236] = {X 454.2197, Y 58.9691, Z -4.6667, A 0.000, B 0.000, C 0.000 }
gfCNCPoint3[26237] = {X 454.2196, Y 58.0000, Z -4.6667, A 0.000, B 0.000, C 0.000 }
gfCNCPoint3[26238] = {X 454.3259, Y 57.0565, Z -4.6667, A 0.000, B 0.000, C 0.000 }
gfCNCPoint3[26239] = {X 454.6395, Y 56.1603, Z -4.6667, A 0.000, B 0.000, C 0.000 }
gfCNCPoint3[26240] = {X 455.1446, Y 55.3564, Z -4.6667, A 0.000, B 0.000, C 0.000 }
gfCNCPoint3[26241] = {X 455.8160, Y 54.6850, Z -4.6667, A 0.000, B 0.000, C 0.000 }
gfCNCPoint3[26242] = {X 456.6199, Y 54.1799, Z -4.6667, A 0.000, B 0.000, C 0.000 }
gfCNCPoint3[26243] = {X 457.5161, Y 53.8663, Z -4.6667, A 0.000, B 0.000, C 0.000 }
gfCNCPoint3[26244] = {X 458.4596, Y 53.7600, Z -4.6667, A 0.000, B 0.000, C 0.000 }
gfCNCPoint3[26245] = {X 475.0000, Y 53.7600, Z -4.6667, A 0.000, B 0.000, C 0.000 }
gfCNCPoint3[26246] = {X 475.9435, Y 53.8663, Z -4.6667, A 0.000, B 0.000, C 0.000 }
gfCNCPoint3[26247] = {X 476.8397, Y 54.1799, Z -4.6667, A 0.000, B 0.000, C 0.000 }
gfCNCPoint3[26248] = {X 477.6436, Y 54.6850, Z -4.6667, A 0.000, B 0.000, C 0.000 }
gfCNCPoint3[26249] = {X 478.3150, Y 55.3564, Z -4.6667, A 0.000, B 0.000, C 0.000 }
gfCNCPoint3[26250] = {X 478.8201, Y 56.1603, Z -4.6667, A 0.000, B 0.000, C 0.000 }
gfCNCPoint3[26251] = {X 479.1337, Y 57.0565, Z -4.6667, A 0.000, B 0.000, C 0.000 }
gfCNCPoint3[26252] = {X 479.2400, Y 58.0000, Z -4.6667, A 0.000, B 0.000, C 0.000 }
gfCNCPoint3[26253] = {X 479.2400, Y 58.9342, Z -4.6667, A 0.000, B 0.000, C 0.000 }
gfCNCPoint3[26254] = {X 479.1496, Y 59.8049, Z -4.6667, A 0.000, B 0.000, C 0.000 }
gfCNCPoint3[26255] = {X 478.8823, Y 60.6385, Z -4.6667, A 0.000, B 0.000, C 0.000 }
gfCNCPoint3[26256] = {X 478.4496, Y 61.3994, Z -4.6667, A 0.000, B 0.000, C 0.000 }
gfCNCPoint3[26257] = {X 477.8698, Y 62.0552, Z -4.6667, A 0.000, B 0.000, C 0.000 }
gfCNCPoint3[26258] = {X 477.1677, Y 62.5780, Z -4.6667, A 0.000, B 0.000, C 0.000 }
gfCNCPoint3[26259] = {X 476.3732, Y 62.9455, Z -4.6667, A 0.000, B 0.000, C 0.000 }
gfCNCPoint3[26260] = {X 475.5202, Y 63.1420, Z -4.6667, A 0.000, B 0.000, C 0.000 }
gfCNCPoint3[26261] = {X 475.5207, Y 92.8325, Z -4.6667, A 0.000, B 0.000, C 0.000 }
gfCNCPoint3[26262] = {X 475.9449, Y 92.9358, Z -4.6667, A 0.000, B 0.000, C 0.000 }
gfCNCPoint3[26263] = {X 476.3628, Y 93.0627, Z -4.6667, A 0.000, B 0.000, C 0.000 }
gfCNCPoint3[26264] = {X 477.1592, Y 93.4247, Z -4.6667, A 0.000, B 0.000, C 0.000 }
gfCNCPoint3[26265] = {X 477.8637, Y 93.9433, Z -4.6667, A 0.000, B 0.000, C 0.000 }
gfCNCPoint3[26266] = {X 478.4458, Y 94.5963, Z -4.6667, A 0.000, B 0.000, C 0.000 }
gfCNCPoint3[26267] = {X 478.8806, Y 95.3555, Z -4.6667, A 0.000, B 0.000, C 0.000 }
gfCNCPoint3[26268] = {X 479.1492, Y 96.1881, Z -4.6667, A 0.000, B 0.000, C 0.000 }
gfCNCPoint3[26269] = {X 479.2400, Y 97.0582, Z -4.6667, A 0.000, B 0.000, C 0.000 }
gfCNCPoint3[26270] = {X 479.2400, Y 98.0000, Z -4.6667, A 0.000, B 0.000, C 0.000 }
gfCNCPoint3[26271] = {X 479.1337, Y 98.9435, Z -4.6667, A 0.000, B 0.000, C 0.000 }
gfCNCPoint3[26272] = {X 478.8201, Y 99.8397, Z -4.6667, A 0.000, B 0.000, C 0.000 }
gfCNCPoint3[26273] = {X 478.3150, Y 100.6436, Z -4.6667, A 0.000, B 0.000, C 0.000 }
gfCNCPoint3[26274] = {X 477.6436, Y 101.3150, Z -4.6667, A 0.000, B 0.000, C 0.000 }
gfCNCPoint3[26275] = {X 476.8397, Y 101.8201, Z -4.6667, A 0.000, B 0.000, C 0.000 }
gfCNCPoint3[26276] = {X 475.9435, Y 102.1337, Z -4.6667, A 0.000, B 0.000, C 0.000 }
gfCNCPoint3[26277] = {X 475.0000, Y 102.2400, Z -4.6667, A 0.000, B 0.000, C 0.000 }
gfCNCPoint3[26278] = {X 458.4596, Y 102.2400, Z -4.6667, A 0.000, B 0.000, C 0.000 }
gfCNCPoint3[26279] = {X 457.5161, Y 102.1337, Z -4.6667, A 0.000, B 0.000, C 0.000 }
gfCNCPoint3[26280] = {X 456.6199, Y 101.8201, Z -4.6667, A 0.000, B 0.000, C 0.000 }
gfCNCPoint3[26281] = {X 455.8160, Y 101.3150, Z -4.6667, A 0.000, B 0.000, C 0.000 }
gfCNCPoint3[26282] = {X 455.1446, Y 100.6436, Z -4.6667, A 0.000, B 0.000, C 0.000 }
gfCNCPoint3[26283] = {X 454.6395, Y 99.8397, Z -4.6667, A 0.000, B 0.000, C 0.000 }
gfCNCPoint3[26284] = {X 454.3259, Y 98.9435, Z -4.6667, A 0.000, B 0.000, C 0.000 }
gfCNCPoint3[26285] = {X 454.2196, Y 98.0000, Z -4.6667, A 0.000, B 0.000, C 0.000 }
gfCNCPoint3[26286] = {X 454.2196, Y 97.0659, Z -4.6667, A 0.000, B 0.000, C 0.000 }
gfCNCPoint3[26287] = {X 454.3099, Y 96.1957, Z -4.6667, A 0.000, B 0.000, C 0.000 }
gfCNCPoint3[26288] = {X 454.5769, Y 95.3624, Z -4.6667, A 0.000, B 0.000, C 0.000 }
gfCNCPoint3[26289] = {X 455.0092, Y 94.6018, Z -4.6667, A 0.000, B 0.000, C 0.000 }
gfCNCPoint3[26290] = {X 455.5884, Y 93.9460, Z -4.6667, A 0.000, B 0.000, C 0.000 }
gfCNCPoint3[26291] = {X 456.2899, Y 93.4231, Z -4.6667, A 0.000, B 0.000, C 0.000 }
gfCNCPoint3[26292] = {X 457.0838, Y 93.0553, Z -4.6667, A 0.000, B 0.000, C 0.000 }
gfCNCPoint3[26293] = {X 457.9363, Y 92.8584, Z -4.6667, A 0.000, B 0.000, C 0.000 }
gfCNCPoint3[26294] = {X 457.9363, Y 85.5404, Z -4.6667, A 0.000, B 0.000, C 0.000 }
gfCNCPoint3[26295] = {X 444.8501, Y 80.4106, Z -4.6667, A 0.000, B 0.000, C 0.000 }
gfCNCPoint3[26296] = {X 419.9432, Y 96.5450, Z -4.6667, A 0.000, B 0.000, C 0.000 }
gfCNCPoint3[26297] = {X 419.9467, Y 97.0651, Z -4.6667, A 0.000, B 0.000, C 0.000 }
gfCNCPoint3[26298] = {X 419.9467, Y 98.0000, Z -4.6667, A 0.000, B 0.000, C 0.000 }
gfCNCPoint3[26299] = {X 419.8404, Y 98.9435, Z -4.6667, A 0.000, B 0.000, C 0.000 }
gfCNCPoint3[26300] = {X 419.5268, Y 99.8397, Z -4.6667, A 0.000, B 0.000, C 0.000 }
gfCNCPoint3[26301] = {X 419.0217, Y 100.6436, Z -4.6667, A 0.000, B 0.000, C 0.000 }
gfCNCPoint3[26302] = {X 418.3503, Y 101.3150, Z -4.6667, A 0.000, B 0.000, C 0.000 }
gfCNCPoint3[26303] = {X 417.5464, Y 101.8201, Z -4.6667, A 0.000, B 0.000, C 0.000 }
gfCNCPoint3[26304] = {X 416.6502, Y 102.1337, Z -4.6667, A 0.000, B 0.000, C 0.000 }
gfCNCPoint3[26305] = {X 415.7067, Y 102.2400, Z -4.6667, A 0.000, B 0.000, C 0.000 }
gfCNCPoint3[26306] = {X 396.4059, Y 102.2400, Z -4.6667, A 0.000, B 0.000, C 0.000 }
gfCNCPoint3[26307] = {X 395.4625, Y 102.1337, Z -4.6667, A 0.000, B 0.000, C 0.000 }
gfCNCPoint3[26308] = {X 394.5663, Y 101.8201, Z -4.6667, A 0.000, B 0.000, C 0.000 }
gfCNCPoint3[26309] = {X 393.7624, Y 101.3150, Z -4.6667, A 0.000, B 0.000, C 0.000 }
gfCNCPoint3[26310] = {X 393.0910, Y 100.6436, Z -4.6667, A 0.000, B 0.000, C 0.000 }
gfCNCPoint3[26311] = {X 392.5858, Y 99.8397, Z -4.6667, A 0.000, B 0.000, C 0.000 }
gfCNCPoint3[26312] = {X 392.2723, Y 98.9435, Z -4.6667, A 0.000, B 0.000, C 0.000 }
gfCNCPoint3[26313] = {X 392.1659, Y 98.0000, Z -4.6667, A 0.000, B 0.000, C 0.000 }
gfCNCPoint3[26314] = {X 392.1659, Y 97.0659, Z -4.6667, A 0.000, B 0.000, C 0.000 }
gfCNCPoint3[26315] = {X 392.2731, Y 96.1188, Z -4.6667, A 0.000, B 0.000, C 0.000 }
gfCNCPoint3[26316] = {X 392.5891, Y 95.2195, Z -4.6667, A 0.000, B 0.000, C 0.000 }
gfCNCPoint3[26317] = {X 393.0980, Y 94.4136, Z -4.6667, A 0.000, B 0.000, C 0.000 }
gfCNCPoint3[26318] = {X 393.7740, Y 93.7417, Z -4.6667, A 0.000, B 0.000, C 0.000 }
gfCNCPoint3[26319] = {X 394.5831, Y 93.2378, Z -4.6667, A 0.000, B 0.000, C 0.000 }
gfCNCPoint3[26320] = {X 395.4843, Y 92.9273, Z -4.6667, A 0.000, B 0.000, C 0.000 }
gfCNCPoint3[26321] = {X 396.4321, Y 92.8260, Z -4.6667, A 0.000, B 0.000, C 0.000 }
gfCNCPoint3[26322] = {X 397.3693, Y 92.7827, Z -4.6667, A 0.000, B 0.000, C 0.000 }
gfCNCPoint3[26323] = {X 398.3033, Y 92.6937, Z -4.6667, A 0.000, B 0.000, C 0.000 }
gfCNCPoint3[26324] = {X 398.9717, Y 92.5316, Z -4.6667, A 0.000, B 0.000, C 0.000 }
gfCNCPoint3[26325] = {X 399.5872, Y 92.2247, Z -4.6667, A 0.000, B 0.000, C 0.000 }
gfCNCPoint3[26326] = {X 413.8423, Y 83.0959, Z -4.6667, A 0.000, B 0.000, C 0.000 }
gfCNCPoint3[26327] = {X 411.6851, Y 79.7274, Z -4.6667, A 0.000, B 0.000, C 0.000 }
gfCNCPoint3[26328] = {X 413.8854, Y 83.1633, Z -4.6667, A 0.000, B 0.000, C 0.000 }
gfCNCPoint3[26329] = {X 428.4049, Y 73.8651, Z -4.6667, A 0.000, B 0.000, C 0.000 }
gfCNCPoint3[26330] = {X 403.8140, Y 64.2169, Z -4.6667, A 0.000, B 0.000, C 0.000 }
gfCNCPoint3[26331] = {X 402.1004, Y 63.6496, Z -4.6667, A 0.000, B 0.000, C 0.000 }
gfCNCPoint3[26332] = {X 400.3349, Y 63.2738, Z -4.6667, A 0.000, B 0.000, C 0.000 }
gfCNCPoint3[26333] = {X 398.5388, Y 63.0940, Z -4.6667, A 0.000, B 0.000, C 0.000 }
gfCNCPoint3[26334] = {X 397.6210, Y 62.9872, Z -4.6667, A 0.000, B 0.000, C 0.000 }
gfCNCPoint3[26335] = {X 396.7494, Y 62.6805, Z -4.6667, A 0.000, B 0.000, C 0.000 }
gfCNCPoint3[26336] = {X 395.9671, Y 62.1889, Z -4.6667, A 0.000, B 0.000, C 0.000 }
gfCNCPoint3[26337] = {X 395.3125, Y 61.5368, Z -4.6667, A 0.000, B 0.000, C 0.000 }
gfCNCPoint3[26338] = {X 394.8180, Y 60.7562, Z -4.6667, A 0.000, B 0.000, C 0.000 }
gfCNCPoint3[26339] = {X 394.5081, Y 59.8858, Z -4.6667, A 0.000, B 0.000, C 0.000 }
gfCNCPoint3[26340] = {X 394.3979, Y 58.9684, Z -4.6667, A 0.000, B 0.000, C 0.000 }
gfCNCPoint3[26341] = {X 394.3977, Y 58.0000, Z -4.6667, A 0.000, B 0.000, C 0.000 }
gfCNCPoint3[26342] = {X 394.5020, Y 57.0743, Z -4.6667, A 0.000, B 0.000, C 0.000 }
gfCNCPoint3[26343] = {X 394.8097, Y 56.1950, Z -4.6667, A 0.000, B 0.000, C 0.000 }
gfCNCPoint3[26344] = {X 395.3053, Y 55.4063, Z -4.6667, A 0.000, B 0.000, C 0.000 }
gfCNCPoint3[26345] = {X 395.9640, Y 54.7476, Z -4.6667, A 0.000, B 0.000, C 0.000 }
gfCNCPoint3[26346] = {X 396.7528, Y 54.2520, Z -4.6667, A 0.000, B 0.000, C 0.000 }
gfCNCPoint3[26347] = {X 397.6320, Y 53.9443, Z -4.6667, A 0.000, B 0.000, C 0.000 }
gfCNCPoint3[26348] = {X 398.5577, Y 53.8400, Z -4.6667, A 0.000, B 0.000, C 0.000 }
gfCNCPoint3[26349] = {X 419.4886, Y 53.8400, Z -4.6667, A 0.000, B 0.000, C 0.000 }
gfCNCPoint3[26350] = {X 420.4143, Y 53.9443, Z -4.6667, A 0.000, B 0.000, C 0.000 }
gfCNCPoint3[26351] = {X 421.2936, Y 54.2520, Z -4.6667, A 0.000, B 0.000, C 0.000 }
gfCNCPoint3[26352] = {X 422.0823, Y 54.7476, Z -4.6667, A 0.000, B 0.000, C 0.000 }
gfCNCPoint3[26353] = {X 422.7410, Y 55.4063, Z -4.6667, A 0.000, B 0.000, C 0.000 }
gfCNCPoint3[26354] = {X 423.2366, Y 56.1950, Z -4.6667, A 0.000, B 0.000, C 0.000 }
gfCNCPoint3[26355] = {X 423.5443, Y 57.0743, Z -4.6667, A 0.000, B 0.000, C 0.000 }
gfCNCPoint3[26356] = {X 423.6486, Y 58.0000, Z -4.6667, A 0.000, B 0.000, C 0.000 }
gfCNCPoint3[26357] = {X 423.6486, Y 58.3415, Z -4.6667, A 0.000, B 0.000, C 0.000 }
gfCNCPoint3[26358] = {X 429.5531, Y 60.6423, Z -4.6667, A 0.000, B 0.000, C 0.000 }
gfCNCPoint3[26359] = {X 458.0186, Y 71.9362, Z -4.6667, A 0.000, B 0.000, C 0.000 }
gfCNCPoint3[26360] = {X 458.0207, Y 63.0709, Z -4.6667, A 0.000, B 0.000, C 0.000 }
gfCNCPoint3[26361] = {X 457.9183, Y 63.0587, Z -4.6667, A 0.000, B 0.000, C 0.000 }
gfCNCPoint3[26362] = {X 457.8162, Y 63.0440, Z -4.6667, A 0.000, B 0.000, C 0.000 }
gfCNCPoint3[26363] = {X 456.8786, Y 62.7819, Z -4.6667, A 0.000, B 0.000, C 0.000 }
gfCNCPoint3[26364] = {X 456.0277, Y 62.3092, Z -4.6667, A 0.000, B 0.000, C 0.000 }
gfCNCPoint3[26365] = {X 455.3099, Y 61.6516, Z -4.6667, A 0.000, B 0.000, C 0.000 }
gfCNCPoint3[26366] = {X 454.7646, Y 60.8452, Z -4.6667, A 0.000, B 0.000, C 0.000 }
gfCNCPoint3[26367] = {X 454.4216, Y 59.9342, Z -4.6667, A 0.000, B 0.000, C 0.000 }
gfCNCPoint3[26368] = {X 454.2997, Y 58.9684, Z -4.6667, A 0.000, B 0.000, C 0.000 }
gfCNCPoint3[26369] = {X 454.2996, Y 58.0000, Z -4.6667, A 0.000, B 0.000, C 0.000 }
gfCNCPoint3[26370] = {X 454.4039, Y 57.0743, Z -4.6667, A 0.000, B 0.000, C 0.000 }
gfCNCPoint3[26371] = {X 454.7116, Y 56.1950, Z -4.6667, A 0.000, B 0.000, C 0.000 }
gfCNCPoint3[26372] = {X 455.2072, Y 55.4063, Z -4.6667, A 0.000, B 0.000, C 0.000 }
gfCNCPoint3[26373] = {X 455.8659, Y 54.7476, Z -4.6667, A 0.000, B 0.000, C 0.000 }
gfCNCPoint3[26374] = {X 456.6546, Y 54.2520, Z -4.6667, A 0.000, B 0.000, C 0.000 }
gfCNCPoint3[26375] = {X 457.5339, Y 53.9443, Z -4.6667, A 0.000, B 0.000, C 0.000 }
gfCNCPoint3[26376] = {X 458.4596, Y 53.8400, Z -4.6667, A 0.000, B 0.000, C 0.000 }
gfCNCPoint3[26377] = {X 475.0000, Y 53.8400, Z -4.6667, A 0.000, B 0.000, C 0.000 }
gfCNCPoint3[26378] = {X 475.9257, Y 53.9443, Z -4.6667, A 0.000, B 0.000, C 0.000 }
gfCNCPoint3[26379] = {X 476.8050, Y 54.2520, Z -4.6667, A 0.000, B 0.000, C 0.000 }
gfCNCPoint3[26380] = {X 477.5937, Y 54.7476, Z -4.6667, A 0.000, B 0.000, C 0.000 }
gfCNCPoint3[26381] = {X 478.2524, Y 55.4063, Z -4.6667, A 0.000, B 0.000, C 0.000 }
gfCNCPoint3[26382] = {X 478.7480, Y 56.1950, Z -4.6667, A 0.000, B 0.000, C 0.000 }
gfCNCPoint3[26383] = {X 479.0557, Y 57.0743, Z -4.6667, A 0.000, B 0.000, C 0.000 }
gfCNCPoint3[26384] = {X 479.1600, Y 58.0000, Z -4.6667, A 0.000, B 0.000, C 0.000 }
gfCNCPoint3[26385] = {X 479.1600, Y 58.9342, Z -4.6667, A 0.000, B 0.000, C 0.000 }
gfCNCPoint3[26386] = {X 479.0692, Y 59.7983, Z -4.6667, A 0.000, B 0.000, C 0.000 }
gfCNCPoint3[26387] = {X 478.8009, Y 60.6248, Z -4.6667, A 0.000, B 0.000, C 0.000 }
gfCNCPoint3[26388] = {X 478.3668, Y 61.3774, Z -4.6667, A 0.000, B 0.000, C 0.000 }
gfCNCPoint3[26389] = {X 477.7858, Y 62.0235, Z -4.6667, A 0.000, B 0.000, C 0.000 }
